// ---- POUs/METS/Common LIB/02_OUTER LIB/Outer FBs/FB_OUTER_ValidationCameraOut.TcPOU
FUNCTION_BLOCK FB_OUTER_ValidationCameraOut
VAR_INPUT
	bDoubleCameraValidationSystemInUse	: BOOL;
	bNewOuterIsProccesing					: BOOL;
	bValidationTimeout						: BOOL;
	bOuterValidation1CameraDone			: BOOL;
	stOuterValidation1CameraStatus	: ST_SCANNER;
	bOuterValidation2CameraDone			: BOOL;
	stOuterValidation2CameraStatus	: ST_SCANNER;

END_VAR
VAR_OUTPUT
	stOuterValidationCameraStatusOut	: ST_SCANNER;
	bOuterValidationDataReady		: BOOL;

END_VAR
VAR
	fbExecute				: R_TRIG;
	aOuterValidationDataReady		: ARRAY [1..2] OF BOOL;
	aCameraNOKStatistic				: ARRAY[1..4] OF INT;
END_VAR

(* rising edge of bExecute *)
fbExecute(CLK:= bNewOuterIsProccesing);

(* move CaseData *)
IF fbExecute.Q = TRUE THEN

	MEMSET(ADR(stOuterValidationCameraStatusOut), 16#00, SIZEOF(stOuterValidationCameraStatusOut));
	bOuterValidationDataReady	:= FALSE;

	aOuterValidationDataReady[1] := FALSE;
	aOuterValidationDataReady[2] := FALSE;
END_IF

IF bOuterValidation1CameraDone OR NOT bDoubleCameraValidationSystemInUse THEN aOuterValidationDataReady[1] := TRUE;	END_IF
IF bOuterValidation2CameraDone THEN aOuterValidationDataReady[2] := TRUE;	END_IF

IF bValidationTimeout	OR
	(bNewOuterIsProccesing AND	aOuterValidationDataReady[1] AND aOuterValidationDataReady[2]) THEN


	IF stOuterValidation1CameraStatus.sImageData.aCodeData[1].strDataString <> '' AND
			 stOuterValidation2CameraStatus.sImageData.aCodeData[1].strDataString = '' THEN

		stOuterValidationCameraStatusOut := stOuterValidation1CameraStatus;

		aCameraNOKStatistic[1] := aCameraNOKStatistic[1] + 1;

	ELSIF stOuterValidation1CameraStatus.sImageData.aCodeData[1].strDataString = '' AND
			 stOuterValidation2CameraStatus.sImageData.aCodeData[1].strDataString <> '' THEN

		stOuterValidationCameraStatusOut := stOuterValidation2CameraStatus;

		aCameraNOKStatistic[2] := aCameraNOKStatistic[2] + 1;

	ELSIF stOuterValidation1CameraStatus.sImageData.aCodeData[1].strDataString <> '' AND
			 stOuterValidation2CameraStatus.sImageData.aCodeData[1].strDataString <> '' AND
			stOuterValidation1CameraStatus.sImageData.aCodeData[1].strDataString = stOuterValidation2CameraStatus.sImageData.aCodeData[1].strDataString THEN

		stOuterValidationCameraStatusOut := stOuterValidation2CameraStatus;

		aCameraNOKStatistic[3] := aCameraNOKStatistic[3] + 1;

	ELSIF stOuterValidation1CameraStatus.sImageData.aCodeData[1].strDataString <> '' AND
			 stOuterValidation2CameraStatus.sImageData.aCodeData[1].strDataString <> '' AND
			stOuterValidation1CameraStatus.sImageData.aCodeData[1].strDataString <> stOuterValidation2CameraStatus.sImageData.aCodeData[1].strDataString THEN

		stOuterValidationCameraStatusOut := stOuterValidation2CameraStatus;
		stOuterValidationCameraStatusOut.sImageData.aCodeData[1].strDataString	:= cCODE_OVERWIRTTEN;

		aCameraNOKStatistic[4] := aCameraNOKStatistic[4] + 1;

	END_IF

	aOuterValidationDataReady[1] := FALSE;
	aOuterValidationDataReady[2] := FALSE;

	bOuterValidationDataReady := TRUE;
END_IF

END_FUNCTION_BLOCK

// ---- POUs/METS/Common LIB/02_OUTER LIB/Outer FBs/FB_OUTER_WriteErrorTable.TcPOU
(* logs data for failed Outers *)
FUNCTION_BLOCK FB_OUTER_WriteErrorTable
VAR_INPUT
	bExecute									: BOOL;			(* set TRUE to scan arrOuterStatus for invalid Outers *)
	bClearData									: BOOL;			(* set TRUE to clear data for invalid Outers *)
	nOpMode									: INT;
	aConfPackCodeInPosition					: ARRAY[1..2] OF T_PACK_Barcode;
	stOuterPackCodeDataNotFound			: ST_RejectItems;
END_VAR
VAR_IN_OUT
	nErrorIndex			: INT;			(* index of Error Outer to be displayed *)
	aOuterStatus			: ARRAY[1..cMAX_OUTER_STATUS_QUEUE] OF ST_OUTER_Status;	(* Outer status array *)
	aErrorOuters			: ARRAY[1..cMAX_OUTER_STATUS_QUEUE] OF ST_OUTER_Status; (* status for last 50 failed Outers *)
END_VAR
VAR_OUTPUT
	bDone				: BOOL;			(* TRUE = OAC action complete *)
	bBusy				: BOOL;			(* TRUE = OAC action in progress *)
	bError				: BOOL;			(* TRUE = OAC action error *)
	nErrorID				: UDINT;		(* error ID *)
	(*bFileInitOK			: BOOL;*)
	nErrorOuters			: UDINT;		(* Outers added to Error list *)
	stErrorOuter			: ST_OUTER_Status; (* last Outer added to arrErrorOuters *)
END_VAR
VAR
	fbExecute				: R_TRIG;
	fbClearData			: R_TRIG;
	eState				: E_OUTER_State;

	nPackIndex			: T_PositiveINT;
	nOuterIndex			: T_PositiveINT;
	(*nMaxOuterIndex		: INT;*)
	nPackStatusIndex		: T_PositiveINT;

	nDupPackChk			: T_PositiveINT;
	nCheckDoubleFail		: T_PositiveINT;
END_VAR

(* monitor bExecute and bClearData for rising edge *)
fbExecute(CLK := bExecute);
fbClearData(CLK := bClearData);

IF fbClearData.Q = TRUE THEN

	(* clear Outer error data *)
	MEMSET(ADR(aErrorOuters), 16#00, SIZEOF(aErrorOuters));
	(*nErrorIndex := 1;*)
END_IF

CASE eState OF

	(* monitor OAC buffer *)
	E_OUTER_IDLE:

		(* rising edge of bExceute *)
		IF fbExecute.Q = TRUE THEN

			(* update outputs *)
			bDone := FALSE;
			bBusy := TRUE;
			bError := FALSE;
			nErrorID := 0;

			(* clear total and reset flag *)
			nErrorOuters := 0;
			(*nMaxOuterIndex := UDINT_TO_INT(SIZEOF(aOuterStatus) / SIZEOF(aOuterStatus[1]));*)


			eState := E_OUTER_SCAN;

		(* bExecute has been reset *)
		ELSIF bExecute = FALSE THEN

			(* reset outputs *)
			bDone := FALSE;
			bBusy := FALSE;
			bError := FALSE;
			nErrorID := 0;
		END_IF


	(* check for Outers that have failed validation *)
	E_OUTER_SCAN:

		(* scan arrStatusArray *)
		FOR nOuterIndex := 1 TO cMAX_OUTER_STATUS_QUEUE DO

			(* CodingAndTrackingMode  > 0 indicates Outer data present *)
			IF aOuterStatus[nOuterIndex].stOACData.CodingAndTrackingMode > 0  AND nOpMode >= 7 THEN

				(* OAC file write error OR validation failed AND data has not been written to ErrorOAC file *)

				(*IF (aOuterStatus[nOuterIndex].nStatus.11  OR aOuterStatus[nOuterIndex].nStatus.13 ) AND NOT aOuterStatus[nOuterIndex].nStatus.14  THEN*)
				IF aOuterStatus[nOuterIndex].nStatus.11 AND NOT aOuterStatus[nOuterIndex].nStatus.14  THEN

					(* update status and log ID for last Outer added *)
					aOuterStatus[nOuterIndex].nStatus.14 := TRUE;

					(* shift arrOACData from [1..49] to [2..50] and move stOACData to arrOACData [1] *)
					MEMMOVE(ADR(aErrorOuters[2]), ADR(aErrorOuters[1]), SIZEOF(aErrorOuters) - SIZEOF(aErrorOuters[1]));
					MEMMOVE(ADR(aErrorOuters[1]), ADR(aOuterStatus[nOuterIndex]), SIZEOF(aErrorOuters[1]));

					IF	aErrorOuters[1].stOACData.OuterRejectID = stOuterPackCodeDataNotFound.nRejectID THEN

						aErrorOuters[1].stOACData.AggregationCodes[1] := aConfPackCodeInPosition[1];
						aErrorOuters[1].stOACData.AggregationCodes[2] := aConfPackCodeInPosition[2];
					END_IF

					(*IF aErrorOuters[1].nStatus.10 AND aErrorOuters[1].nStatus.13 THEN
						aErrorOuters[1].stOACData.OuterRejectCode	:= CONCAT(aErrorOuters[1].stOACData.OuterRejectCode, ' - OAC File Write Error');
					END_IF*)

					(* update counter and set flag to update error file *)
					stErrorOuter := aErrorOuters[1];
					nErrorOuters := nErrorOuters + 1;

					(*AS mod test for previous existence of the failed outer with the same code(s) failed*)
					(*only check if a pack code is missing!*)
					nCheckDoubleFail := 0;
					FOR nPackIndex := 1 TO cMAX_PACKS_PER_OUTER DO
						IF aErrorOuters[1].stOACData.PackCode[nPackIndex] = '' THEN
							nCheckDoubleFail := nCheckDoubleFail+1;
						END_IF
					END_FOR
					IF (nCheckDoubleFail > 0) AND (nCheckDoubleFail < aErrorOuters[1].stOACData.NumberOfPacks) AND nOpMode = 11 AND NOT(aErrorOuters[1].nStatus.15) THEN
						FOR nDupPackChk := 2 TO cMAX_OUTER_STATUS_QUEUE DO
							FOR nPackStatusIndex :=1 TO cMAX_PACKS_PER_OUTER DO
								IF aErrorOuters[1].stOACData.PackCode[nPackStatusIndex] = aErrorOuters[nDupPackChk].stOACData.PackCode[nPackStatusIndex] THEN
										(*Using status 15 for signifying that an outer has failed more than once for the same reason*)
										aErrorOuters[1].nStatus.15 := TRUE;
										aErrorOuters[nDupPackChk].nStatus.15 := TRUE;
									EXIT;
								END_IF
							END_FOR
						END_FOR
					END_IF

					(* update nErrorIndex so that it moves with Outer if new data is added to arrErrorOuter *)
					nErrorIndex := nErrorIndex + 1;
					EXIT;
				END_IF
			END_IF
		END_FOR

		(* end of arrOuterStatus reached *)
		IF nOuterIndex > cMAX_OUTER_STATUS_QUEUE THEN

			eState := E_OUTER_DONE;

		ELSE

			eState := E_OUTER_SCAN;

		END_IF

	(* OAC file complete *)
	E_OUTER_DONE:

		(* update outputs *)
		bDone := TRUE;
		bBusy := FALSE;

		eState := E_OUTER_IDLE;


(* unknown state *)
ELSE

	eState := E_OUTER_IDLE;

	(* reset outputs *)
	bDone := TRUE;
	bBusy := FALSE;
	bError := TRUE;
	nErrorID := 16#FFFFFFFF;

END_CASE

END_FUNCTION_BLOCK

// ---- POUs/METS/Common LIB/02_OUTER LIB/Outer FBs/FB_OUTER_WriteOACLoopDB.TcPOU
(* scan and validate Outers, generate OAC file for new valid Outers *)
FUNCTION_BLOCK FB_OUTER_WriteOACLoopDB
VAR_INPUT
	bExecute					: BOOL;			(* scan for completed Outer *)
	nPacksPerOuter			: INT;
	bExtendedDupCheck		: BOOL;
	nCodingAndTrackingMode	: INT;
	stCTDateTime				: ST_SYSTEM_DateTime;
END_VAR
VAR_IN_OUT
	stOACDataDB					: ST_DB_OACDataCtrl;
	stLastOACDataDB				: ST_DB_OACDataCtrl;
	stCodeInfo_Pack				: ST_CodeInfo;
	stCodeInfo_Outer			: ST_CodeInfo;
	aOuterStatus				: ARRAY[1..cMAX_OUTER_STATUS_QUEUE] OF ST_OUTER_Status;	(* Outer status array *)
	stLastOuterStatus			: ST_OUTER_Status;
	stOuterDataNotFound			: ST_RejectItems;
	stInfeedQueue				: ST_CASE_InfeedQueue;	(* Infeed Conveyor queue *)
END_VAR
VAR_OUTPUT
	bDone				: BOOL;			(* TRUE = validation complete *)
	bBusy				: BOOL;			(* TRUE = validation in progress *)
	bError				: BOOL;			(* TRUE = validation error *)
	nErrorID				: UDINT;		(* error ID *)
	sOACRecordDBName			: T_MaxString;
	stOuterStatus			: ST_OUTER_Status;	(* Outer status *)
	bOACUpdated			: BOOL;
	sCodesAggregatedToOAC	: T_LongSTRING;
END_VAR
VAR
	fbExecute				: R_TRIG;
	tonTimeOut				: TON;
	rtTimeOutExec				: R_TRIG;

	eState					: E_OUTER_State;
	eErrorState					: E_OUTER_State;
	//nMaxOuterIndex		: INT;
	nOuterIndex			: INT;
	nSourceIndex			: INT;
	nInfeedIndex			: INT;

	nCheckIndex : T_PositiveINT;
	nPackIndex : T_PositiveINT;

	eCodeAIType			: E_CodeAIType;

	sBarcode				: T_OUTER_Barcode;

	nOACDataCreated 			: UDINT;
	nOACStoredInDB 			: UDINT;
	nOACFaildInDB				: UDINT;
	nOACUpdatedInDB			: UDINT;

	aDiagOACDataDB				: ARRAY[0..1] OF ST_DB_OACDataCtrl;

	aLocalOuterStatus			: ARRAY[1..10] OF  ST_OUTER_Status;
	nCounter :UDINT;

	nOACLogIndex			: T_PositiveINT;
	sAppendedString				: STRING;
END_VAR

(***************************************TimeOut *******************************************)
(* monitor Busy timeout *)
tonTimeOut( IN:=nSourceIndex <> 0, PT:=cONE_SECOND, Q=>);

rtTimeOutExec(CLK:= tonTimeOut.Q);

IF rtTimeOutExec.Q THEN

	bError := TRUE;
	nErrorID := 100;
	IF nSourceIndex > 0 THEN

		aOuterStatus[nSourceIndex].sDataSourceTracker 	:= 	'TIMEOUT';
		aOuterStatus[nSourceIndex].nStatus.13 := TRUE;

		stLastOuterStatus := aOuterStatus[nSourceIndex];

		sCodesAggregatedToOAC	:= 'TIMEOUT_OUT';
		bOACUpdated	:= TRUE;

	END_IF

	MEMSET(ADR(stOACDataDB), 16#00, SIZEOF(stOACDataDB));
	MEMSET(ADR(stLastOACDataDB), 16#00, SIZEOF(stLastOACDataDB));


	eState := E_OUTER_DONE;
END_IF

(***************************************Execution*******************************************)

(* monitor rising edge of bExecute *)
fbExecute(CLK := bExecute);

(* rising edge of bExecute *)
CASE eState OF

	(* idle *)
	E_OUTER_IDLE:

		(* scan for completed Outer when OAC files are required *)
		IF fbExecute.Q = TRUE THEN

			(* update outputs *)
			bDone := FALSE;
			bBusy := TRUE;
			bError := FALSE;
			nErrorID := 0;

			(* clear outputs *)
			nOACDataCreated 		:= 0;
			nOACStoredInDB 		:= 0;
			nOACFaildInDB			:= 0;

			(* max Outer index *)
			//nMaxOuterIndex := UDINT_TO_INT(SIZEOF(aOuterStatus) / SIZEOF(aOuterStatus[1]));

			eState := E_OUTER_SCAN;

		(* no action required *)
		ELSIF bExecute = FALSE THEN

			(* reset outputs *)
			bDone := FALSE;
			bBusy := FALSE;
			bError := FALSE;
			nErrorID := 0;
		END_IF


	(* scan for completed Outer *)
	E_OUTER_SCAN:

		(* reset index of Outer to be written to OAC file *)
		nSourceIndex 			:= 0;

		sBarcode					:= '';
		bOACUpdated				:= FALSE;

		(* scan aOuterStatus  backward - ensures that oldest Outer will be written first *)
		FOR nOuterIndex := cMAX_OUTER_STATUS_QUEUE TO 1 BY -1 DO

			(* TriggerID > 0 indicates Outer data present -  *)
			IF aOuterStatus[nOuterIndex].nTriggerID > 0 AND
				aOuterStatus[nOuterIndex].stOACData.CodingAndTrackingMode >= 7 AND
				(aOuterStatus[nOuterIndex].nStatus.10  OR
					(aOuterStatus[nOuterIndex].nStatus.11 AND aOuterStatus[nOuterIndex].nStatus.14)) AND
				NOT aOuterStatus[nOuterIndex].nStatus.12 AND
				NOT aOuterStatus[nOuterIndex].nStatus.13 THEN

				(* log index of Outer requiring OAC file *)
				nSourceIndex := nOuterIndex;
				EXIT;
			END_IF
		END_FOR

		(* Outer found requiring OAC file to be written *)
		IF nSourceIndex > 0 THEN

			(* copy Outer data from aOuterStatus *)
			stOuterStatus := aOuterStatus[nSourceIndex];

			nOACDataCreated := nOACDataCreated +1;

			IF	bExtendedDupCheck AND aOuterStatus[nSourceIndex+1].nStatus.12 AND nSourceIndex <  cMAX_OUTER_STATUS_QUEUE  THEN
				(* for all other Packs in Outer *)
				FOR  nPackIndex :=1 TO cMAX_PACKS_PER_OUTER DO
	
					IF stOuterStatus.stOACData.PackCodeStatus[nPackIndex].5 OR stOuterStatus.stOACData.PackCodeStatus[nPackIndex].6 THEN

						FOR nCheckIndex :=1 TO cMAX_PACKS_PER_OUTER DO

							IF stOuterStatus.stOACData.PackCode[nPackIndex] = aOuterStatus[nSourceIndex+1].stOACData.PackCode[nCheckIndex] THEN

								stOuterStatus.nStatus.22 := TRUE;
								stOuterStatus.sDataSourceTracker  := 'OUT_DUPLIC';

								aOuterStatus[nSourceIndex+1].nStatus.22 := TRUE;
								aOuterStatus[nSourceIndex+1].sDataSourceTracker  := 'OUT_DUPLIC';

								EXIT;
							END_IF
						END_FOR
						EXIT;
					END_IF
				END_FOR
			END_IF

			IF aOuterStatus[nSourceIndex+1].nStatus.22 AND stOuterStatus.nStatus.22  AND nSourceIndex <  cMAX_OUTER_STATUS_QUEUE  THEN

				FOR nInfeedIndex:=1 TO stInfeedQueue.nIndex DO 
					IF stInfeedQueue.aOuter[nInfeedIndex].Barcode = aOuterStatus[nSourceIndex+1].stOACData.Barcode 	AND 
						aOuterStatus[nSourceIndex+1].stOACData.Barcode <> ''				 						THEN
						
						stInfeedQueue.aOuter[nInfeedIndex].DataSource 		:= 'B_22';
						stInfeedQueue.aOuter[nInfeedIndex].OuterRejectCode 	:= stOuterDataNotFound.sMetsDisplayCode;
						stInfeedQueue.aOuter[nInfeedIndex].OuterRejectID	:= stOuterDataNotFound.nRejectID;
					END_IF
				END_FOR
				
				stLastOACDataDB.stOACStatusDB	:= aOuterStatus[nSourceIndex+1];
				stLastOACDataDB.bBlockRecord	:= TRUE;
				stLastOACDataDB.bUpdateDataReq 	:= TRUE;

				eState := E_OUTER_UPDATEDATA;
			ELSE
				eState := E_OUTER_WRITEDATA;
			END_IF
		ELSE
			eState := E_OUTER_DONE;
		END_IF

	E_OUTER_UPDATEDATA:

		IF	stLastOACDataDB.bDone	THEN

			IF NOT  stLastOACDataDB.bError THEN

				nOACUpdatedInDB := nOACUpdatedInDB +1;
			ELSE
				bError := TRUE;
				nErrorID := stLastOACDataDB.nErrorID;
				eErrorState := eState;
			END_IF

			aDiagOACDataDB[1]	:= stLastOACDataDB;

			eState := E_OUTER_WRITEDATA;
		END_IF


	E_OUTER_WRITEDATA:

		IF F_InvalidateASCIIChar(F_CODE_GetItem(stOuterStatus.stOACData.Barcode, eCodeAIType.SerialCode, stCodeInfo_Outer)) >	0 	THEN

			stOuterStatus.sDataSourceTracker  := 'BRCD_INVAL';
			stOuterStatus.nStatus.22 := TRUE;
		ELSE
			stOACDataDB.sFileCodeName	:= F_CodeToHex(F_CODE_GetItem(stOuterStatus.stOACData.Barcode , eCodeAIType.SerialCode, stCodeInfo_Outer));
		END_IF

		IF stOuterStatus.nStatus.22 THEN
			stOACDataDB.bBlockRecord		:= TRUE;
		END_IF
		stOACDataDB.stOACStatusDB			:= stOuterStatus;
		stOACDataDB.bCreateDataReq			:= TRUE;

(*place for HectorDB block*)

		IF	stOACDataDB.bDone	THEN

			sOACRecordDBName	:= stOACDataDB.sFileCodeName;

			IF NOT  stOACDataDB.bError THEN

				(* count OAC records stored *)
				nOACStoredInDB := nOACStoredInDB + 1;
				(* update sOuterStatus - OAC record written OK *)
				stOuterStatus.nStatus.12 := TRUE;

			ELSE
				bError := TRUE;
				nErrorID := stOACDataDB.nErrorID;
				nOACFaildInDB := nOACFaildInDB + 1;
				(* update sOuterStatus - OAC file write error *)
				stOuterStatus.stOACData.OuterCodeStatus.6 := TRUE;
				stOuterStatus.nStatus.13 := TRUE;
				eErrorState := eState;
			END_IF

			aDiagOACDataDB[0]	:= stOACDataDB;

			eState := E_OUTER_UPDATESTATUS;

		END_IF

	(* update Outer status *)
	E_OUTER_UPDATESTATUS:

		MEMSET(ADR(stOACDataDB), 16#00, SIZEOF(stOACDataDB));		(*or moved to te execution part at the begining*)
		MEMSET(ADR(stLastOACDataDB), 16#00, SIZEOF(stLastOACDataDB));		(*or moved to te execution part at the begining*)

		(* move stOuterStatus data back to shift reg *)
		FOR nOuterIndex := cMAX_OUTER_STATUS_QUEUE TO 1 BY -1 DO

			(* matching nTriggerID found *)
			IF aOuterStatus[nOuterIndex].nTriggerID = stOuterStatus.nTriggerID AND
				NOT aOuterStatus[nOuterIndex].nStatus.12 AND NOT aOuterStatus[nOuterIndex].nStatus.13 THEN


				nCounter := nCounter +1;
		(*!*)	stLastOuterStatus :=stOuterStatus;
				MEMMOVE(ADR(aLocalOuterStatus[2]), ADR(aLocalOuterStatus[1]), SIZEOF(aLocalOuterStatus)-SIZEOF(aLocalOuterStatus[1]));
				aLocalOuterStatus[1] :=stLastOuterStatus;

				(* move updated Outer data to shift reg *)
				aOuterStatus[nOuterIndex] := stOuterStatus;

				sAppendedString			:= '';
				sCodesAggregatedToOAC	:= '';
				
				sCodesAggregatedToOAC := F_CONCAT3(aOuterStatus[nOuterIndex].stOACData.OuterRejectCode,' - ',  F_CODE_GetItem(aOuterStatus[nOuterIndex].stOACData.Barcode, eCodeAIType.SerialCode, stCodeInfo_Outer));
				sCodesAggregatedToOAC := F_CONCAT6(sCodesAggregatedToOAC,'	[', RIGHT(aOuterStatus[nOuterIndex].stOACData.AggregationCodes[1],7),']:[',RIGHT(aOuterStatus[nOuterIndex] .stOACData.AggregationCodes[2],7),']');

				FOR nOACLogIndex := 1 TO MIN(nPacksPerOuter ,cMAX_PACKS_PER_OUTER) BY 1 DO
					//sCodesAggregatedToOAC :=F_LongCONCAT(sCodesAggregatedToOAC, '     ');
					//sCodesAggregatedToOAC := F_LongCONCAT(sCodesAggregatedToOAC, RIGHT(F_CODE_GetItem(aOuterStatus[nOuterIndex] .stOACData.PackCode[nOACLogIndex], eCodeAIType.SerialCode, stCodeInfo_Pack),7));
				
					CONCAT2(ADR(sCodesAggregatedToOAC), ADR('   '), ADR(sCodesAggregatedToOAC), SIZEOF(sCodesAggregatedToOAC));
		
					sAppendedString := RIGHT(F_CODE_GetItem(aOuterStatus[nOuterIndex].stOACData.PackCode[nOACLogIndex], eCodeAIType.SerialCode, stCodeInfo_Pack),7);
					CONCAT2(ADR(sCodesAggregatedToOAC), ADR(sAppendedString), ADR(sCodesAggregatedToOAC), SIZEOF(sCodesAggregatedToOAC));

				END_FOR

				bOACUpdated := TRUE;
				EXIT;
			END_IF
		END_FOR

		eState := E_OUTER_SCAN;

	(* OAC file complete *)
	E_OUTER_DONE:

		(* update outputs *)
		bDone := TRUE;
		bBusy := FALSE;

		eState := E_OUTER_IDLE;


(* unknown state *)
ELSE

	eState := E_OUTER_IDLE;
END_CASE

END_FUNCTION_BLOCK

// ---- POUs/METS/Common LIB/02_OUTER LIB/Outer Functions/F_OUTER_GetRejectReasonFSS.TcPOU
FUNCTION F_OUTER_GetRejectReasonFSS : T_FSS_RejecCode
VAR_INPUT
	sRejectReasonME			:	STRING(255);
	stOuterRejectReasons	: ST_RejectReasonsForOuter;
END_VAR
VAR
	sRejectReasonFSS:	T_FSS_RejecCode;
END_VAR

IF sRejectReasonME = 'OK' THEN
	sRejectReasonFSS := '';

ELSIF sRejectReasonME = '' THEN
	sRejectReasonFSS := stOuterRejectReasons.stUnknownOuterReject.sFssSendCode;

ELSIF FIND(sRejectReasonME, stOuterRejectReasons.stOuterBarcodeGtinError.sMetsSearchCode) > 0 THEN
	sRejectReasonFSS := stOuterRejectReasons.stOuterBarcodeGtinError.sFssSendCode;

ELSIF FIND(sRejectReasonME, stOuterRejectReasons.stOuterBarcodeRskuError.sMetsSearchCode) > 0 THEN
	sRejectReasonFSS := stOuterRejectReasons.stOuterBarcodeRskuError.sFssSendCode;

ELSIF FIND(sRejectReasonME, stOuterRejectReasons.stOuterCodeSerialError.sMetsSearchCode) > 0 THEN
	sRejectReasonFSS := stOuterRejectReasons.stOuterCodeSerialError.sFssSendCode;

ELSIF FIND(sRejectReasonME, stOuterRejectReasons.stOuterBarcodeInvalidLength.sMetsSearchCode) > 0 THEN
	sRejectReasonFSS := stOuterRejectReasons.stOuterBarcodeInvalidLength.sFssSendCode;

ELSIF FIND(sRejectReasonME, stOuterRejectReasons.stOuterBarcodeNotRead.sMetsSearchCode) > 0 THEN
	sRejectReasonFSS := stOuterRejectReasons.stOuterBarcodeNotRead.sFssSendCode;

ELSIF FIND(sRejectReasonME, stOuterRejectReasons.stOuterBarcodeDuplicate.sMetsSearchCode) > 0 THEN
	sRejectReasonFSS := stOuterRejectReasons.stOuterBarcodeDuplicate.sFssSendCode;

ELSIF FIND(sRejectReasonME,stOuterRejectReasons.stOuterDataNotFound.sMetsSearchCode) > 0 THEN
	sRejectReasonFSS := stOuterRejectReasons.stOuterDataNotFound.sFssSendCode;

ELSIF FIND(sRejectReasonME, stOuterRejectReasons.stOuterGeneralCodeError.sMetsSearchCode) > 0 THEN
	sRejectReasonFSS := stOuterRejectReasons.stOuterGeneralCodeError.sFssSendCode;

ELSIF FIND(sRejectReasonME, stOuterRejectReasons.stOuterTimeOutValidation.sMetsSearchCode) > 0 THEN
	sRejectReasonFSS := stOuterRejectReasons.stOuterTimeOutValidation.sFssSendCode;

ELSIF FIND(sRejectReasonME, stOuterRejectReasons.stOuterDuplicatedPackCodesFound.sMetsSearchCode) > 0 THEN
	sRejectReasonFSS := stOuterRejectReasons.stOuterDuplicatedPackCodesFound.sFssSendCode;

ELSIF FIND(sRejectReasonME, stOuterRejectReasons.stOuterPackCodeDataNotFound.sMetsSearchCode) > 0 THEN
	sRejectReasonFSS := stOuterRejectReasons.stOuterPackCodeDataNotFound.sFssSendCode;

ELSIF FIND(sRejectReasonME, stOuterRejectReasons.stOuterConfirmCodeNotRead.sMetsSearchCode) > 0 THEN
	sRejectReasonFSS := stOuterRejectReasons.stOuterConfirmCodeNotRead.sFssSendCode;

ELSIF FIND(sRejectReasonME, stOuterRejectReasons.stOuterPackCodeInvalid.sMetsSearchCode) > 0 THEN
	sRejectReasonFSS := stOuterRejectReasons.stOuterPackCodeInvalid.sFssSendCode;

ELSIF FIND(sRejectReasonME, stOuterRejectReasons.stOuterPackCodeNotRead.sMetsSearchCode) > 0 THEN
	sRejectReasonFSS := stOuterRejectReasons.stOuterPackCodeNotRead.sFssSendCode;

ELSIF FIND(sRejectReasonME, stOuterRejectReasons.stOuterQAReject.sMetsSearchCode) > 0 THEN
	sRejectReasonFSS := stOuterRejectReasons.stOuterQAReject.sFssSendCode;

ELSIF FIND(sRejectReasonME, stOuterRejectReasons.stOuterPackCodeDBError.sMetsSearchCode) > 0 THEN
	sRejectReasonFSS := stOuterRejectReasons.stOuterPackCodeDBError.sFssSendCode;

ELSIF FIND(sRejectReasonME, stOuterRejectReasons.stOuterBarcodeDBError.sMetsSearchCode) > 0 THEN
	sRejectReasonFSS := stOuterRejectReasons.stOuterBarcodeDBError.sFssSendCode;

ELSIF FIND(sRejectReasonME, stOuterRejectReasons.stOuterCodesBrandSpecError.sMetsSearchCode) > 0 THEN
	sRejectReasonFSS := stOuterRejectReasons.stOuterCodesBrandSpecError.sFssSendCode;

ELSE
	sRejectReasonFSS := stOuterRejectReasons.stUnknownOuterReject.sFssSendCode;
END_IF

F_OUTER_GetRejectReasonFSS := sRejectReasonFSS;

END_FUNCTION

// ---- POUs/METS/Common LIB/02_OUTER LIB/Outer Functions/F_OUTER_HexToBarcode.TcPOU
FUNCTION F_OUTER_HexToBarcode : STRING(255)
VAR_INPUT
	strSerialCodeInHex	: STRING(255);
END_VAR
VAR

	nBarcodeLen		: INT;
	nCharIndex		: INT;
	strCharInHex			: STRING(2);
	nAsciiCode			:BYTE;
	strChar			: STRING(2);
END_VAR

(* reset output *)
F_OUTER_HexToBarcode := '';

(* length of strPackCode *)
nBarcodeLen := LEN(strSerialCodeInHex);

(* strPackCode contains data *)
IF nBarcodeLen > 0 THEN

	(* check each char in the code *)
	FOR nCharIndex := 1 TO nBarcodeLen BY 2 DO

		(* get char from string *)
		strCharInHex := MID(strSerialCodeInHex, 2, nCharIndex);
		HEXSTR_TO_DATA(strCharInHex, ADR(nAsciiCode), SIZEOF(nAsciiCode));
		strChar := F_ToCHR(nAsciiCode);
		F_OUTER_HexToBarcode := CONCAT(F_OUTER_HexToBarcode, strChar);
	END_FOR
END_IF

END_FUNCTION

// ---- POUs/METS/Common LIB/02_OUTER LIB/Outer Functions/F_OUTER_ProgNumberMap.TcPOU
FUNCTION F_OUTER_ProgNumberMap : BOOL

VAR
	nPackIndex			: INT;
END_VAR
(*All VAR_IN_OUT variables have been moved to the end of the declaration due to compatibility reasons*)
VAR_IN_OUT
	stImageData				: ST_SCANNER_ImageData;	(* scanner response data *)
END_VAR

FOR nPackIndex := 1 TO LIMIT(1, stImageData.nCodesRead, cMAX_CAMERA_PROG_NUMBER) DO

	IF stImageData.aCodeData[nPackIndex].nProgramNo = 0 THEN

		(* code is in upper left quadrant of image *)
		IF stImageData.aCodeData[nPackIndex].fXPos >= 0 THEN

			(* get pack position within Outer *)
			stImageData.aCodeData[nPackIndex].nProgramNo := 1;

		(* code is in lower left quadrant of image *)
		ELSIF stImageData.aCodeData[nPackIndex].fXPos < 0 THEN

			(* get pack position within Outer *)
			stImageData.aCodeData[nPackIndex].nProgramNo := 2;
		END_IF
	END_IF
END_FOR

END_FUNCTION

// ---- POUs/METS/Common LIB/04_CASE LIB/Case FBs/FB_CASE_AddOACDataDBLoop.TcPOU
FUNCTION_BLOCK FB_CASE_AddOACDataDBLoop
VAR_INPUT
	bExecute					: BOOL;			(* scan for valid Outer in arrOuterStatus *)
	bStopOnInvalidCode		: BOOL;						(* set TRUE to give alarm if an invalid code is detected *)
	//bFileReadOnly				: BOOL;
	bATTPModeEnable			: BOOL;
	//sLocalOACPath				: T_FolderPath;	(* TEMP folder path *)
	stCTDateTime				: ST_SYSTEM_DateTime;	(* CaseTrace date/time structure *)
	stOuterDataNotFound		: ST_RejectItems;
END_VAR
VAR_IN_OUT
	stOACDataDB					: ST_DB_OACDataCtrl;
	stCodeInfo_Outer			: ST_CodeInfo;
	stProductInstruction			: ST_PCM_Status;
	aOuterStatus				: ARRAY[1..cMAX_OUTER_STATUS_QUEUE] OF ST_OUTER_Status;	(* Outer status array *)
	stInfeedQueue				: ST_CASE_InfeedQueue;	(* Infeed Conveyor queue *)
END_VAR
VAR_OUTPUT
	bDone					: BOOL;			(* TRUE = write OAC file complete *)
	bBusy					: BOOL;			(* TRUE = write OAC file in progress *)
	bError					: BOOL;			(* TRUE = write OAC file error *)
	nErrorID					: UDINT;			(* error ID *)

	nOACFilesRead				: UDINT;
	nReadOACDataFromStructure	: INT;
	nReadOACDataFromFile		: INT;
	nOACFilesFalseRead 		: INT;

	sOACFile					: T_OAC_Filename;
	stOACData				: ST_OAC_Data;
	bScaningActive			: BOOL;
END_VAR
VAR
	fbExecute					: R_TRIG;
	eState					: E_CASE_State;
	eErrorState				: E_CASE_State;
	nOuterIndex				: INT;
	nMaxOuterIndex			: INT;

	sCurrnetInfeedBarcode		: T_MaxString;
	fbReadXMLData			: FB_XmlSrvRead;
	nScanIndex				: INT;

	sOuterTimeStamp				: T_ISO8601Time;
	bOuterMasterListRestored	: BOOL;
	sDataSource				: STRING(4);

	nCounter					: INT;
END_VAR

(* monitor bExecute for rising edge *)
fbExecute(CLK := bExecute);

CASE eState OF

	(* idle state *)
	E_CASE_IDLE:

		(* rising edge of bExecute *)
		IF fbExecute.Q = TRUE THEN

			(* update outputs *)
			bDone := FALSE;
			bBusy := TRUE;
			bError := FALSE;
			nErrorID := 0;

			(* clear outputs *)
			nOACFilesRead := 0;
			sOACFile := '';
			(*MEMSET(ADR(stOACData), 16#00, SIZEOF(stOACData));*)
			sDataSource :='';
			nMaxOuterIndex := UDINT_TO_INT(SIZEOF(aOuterStatus) / SIZEOF(aOuterStatus[1]));

			(*nOuterIndex := 1;*)

			eState := E_CASE_SCANINFEEDQUEUE;

		(* OAC data disabled *)
		ELSIF bExecute = FALSE THEN

			(* reset outputs *)
			bDone := FALSE;
			bBusy := FALSE;
			bError := FALSE;
			nErrorID := 0;

			bScaningActive := FALSE;

		END_IF


	(* scan for missing OAC data *)
	E_CASE_SCANINFEEDQUEUE:

		(* preset next state, will be udpated if an Outer without OAC data is found in Infeed Queue *)
		MEMSET(ADR(stOACData), 16#00, SIZEOF(stOACData));
		eState := E_CASE_DONE;

		(* scan remainder of Infeed Queue *)
		FOR nScanIndex := 1 TO  MIN(stInfeedQueue.nIndex, cMAX_INFEED_QUEUE) DO

			(* OAC data has not been read *)
			IF stInfeedQueue.aOuter[nScanIndex].CodingAndTrackingMode = 0 AND  stInfeedQueue.aOuter[nScanIndex].DataSource = '' THEN

				IF (*stProductInstruction.nOpMode = 7 AND*) NOT stProductInstruction.bEnablePacks (*AND bStopOnInvalidCode*) THEN
					stInfeedQueue.aOuter[nScanIndex].ProductionDate := F_StringWildcard('#YYYYMMDD#', stCTDateTime.sSystemTime);
					stInfeedQueue.aOuter[nScanIndex].ProductionTime := F_StringWildcard('#hhmmss#', stCTDateTime.sSystemTime);
					stInfeedQueue.aOuter[nScanIndex].ProductionTimeOffset := F_SYSTEM_SystemTimeOffsetToHHMM(stCTDateTime.nSystemTimeOffset);

					stInfeedQueue.aOuter[nScanIndex].OuterTimeStamp :=F_SYSTEM_SystemTimeAsISO8601(stCTDateTime.sSystemTime, stCTDateTime.sUTCTimeZoneOffset );
					stInfeedQueue.aOuter[nScanIndex].RetailSKU := stProductInstruction.sRetailSKU;
					stInfeedQueue.aOuter[nScanIndex].OuterMachine.ProductionSite :=  stProductInstruction.sProductionSite;
					stInfeedQueue.aOuter[nScanIndex].OuterMachine.ProductionLine := stProductInstruction.sProductionLine;
					stInfeedQueue.aOuter[nScanIndex].BatchNumber := stProductInstruction.sBatchNumber;
					stInfeedQueue.aOuter[nScanIndex].CodingAndTrackingMode := stProductInstruction.nOpMode;

					stInfeedQueue.aOuter[nScanIndex].DataSource := 'REST';
					stInfeedQueue.aOuter[nScanIndex].OuterRejectCode := 'OK';
					stInfeedQueue.aOuter[nScanIndex].OuterRejectID := 0;

					eState := E_CASE_SCANINFEEDQUEUE;

				ELSE
					sCurrnetInfeedBarcode 	:=	 stInfeedQueue.aOuter[nScanIndex].Barcode ;
					bOuterMasterListRestored 	:= stInfeedQueue.aOuter[nScanIndex].OuterMasterListRestored;
					(*sOuterTimeStamp			:= stInfeedQueue.aOuter[nScanIndex].OuterTimeStamp;*)
					sDataSource :='';
					(* generate OAC file name and clear data for last OAC file *)

					(*sOACFile := F_CONCAT3('OAC_', F_OUTER_BarcodeToHex(sCurrnetInfeedBarcode), '.xml');*)

					IF bTempBlockReadFromStruct THEN
						eState := E_CASE_SCANOUTERS;
					ELSE
						eState := E_CASE_READOACDATA;
					END_IF
				END_IF

				bScaningActive := TRUE;
				EXIT;
			END_IF
		END_FOR

	E_CASE_SCANOUTERS:


		FOR nOuterIndex := 1 TO nMaxOuterIndex DO

			(* TriggerID > 0 indicates Outer data present *)
			IF	 aOuterStatus[nOuterIndex].bLabelApplied 
				AND NOT aOuterStatus[nOuterIndex].nStatus.19 
				AND NOT aOuterStatus[nOuterIndex].nStatus.22 THEN

				IF  aOuterStatus[nOuterIndex].stOACData.Barcode = sCurrnetInfeedBarcode  THEN

					stOACData	 := aOuterStatus[nOuterIndex].stOACData;
					EXIT;
				END_IF
			END_IF
		END_FOR

		IF stOACData.CodingAndTrackingMode > 0 OR stOACData.OuterRejectCode <> '' THEN

			nOACFilesRead := nOACFilesRead + 1;
			sDataSource := 'ST';
			nReadOACDataFromStructure:= nReadOACDataFromStructure + 1;

			eState := E_CASE_UPDATEINFEEDQUEUE;
		ELSE
			eState := E_CASE_READOACDATA;
		END_IF

	(* read data from OAC *)
	E_CASE_READOACDATA:

				stOACDataDB.bReadDataReq		:=TRUE;

				(*stOACDataDB.sFileCodeName		 := F_OUTER_BarcodeToHex(sCurrnetInfeedBarcode);*)

				IF F_InvalidateASCIIChar(F_CODE_GetItem(sCurrnetInfeedBarcode, eCodeAIType.SerialCode, stCodeInfo_Outer)) >	0 	THEN
		
					stOACDataDB.sFileCodeName := '';
				ELSE
					stOACDataDB.sFileCodeName	:= F_CodeToHex(F_CODE_GetItem(sCurrnetInfeedBarcode , eCodeAIType.SerialCode, stCodeInfo_Outer));
				END_IF

				IF stOACDataDB.bDone THEN
					IF NOT stOACDataDB.bError THEN		(* f.ex not found, or DB transaction faild??*)

						IF NOT  stOACDataDB.stOACStatusDB.nStatus.22 THEN

							stOACData := stOACDataDB.stOACStatusDB.stOACData;
							sDataSource := 'DB';
						ELSE
							sDataSource := 'B_22';
						END_IF

						nOACFilesRead := nOACFilesRead + 1;

					ELSE
						bError := TRUE;
						nErrorID := stOACDataDB.nErrorID;
						sDataSource := 'NO_R';

						eErrorState := eState;
					END_IF

					eState := E_CASE_UPDATEINFEEDQUEUE;

				END_IF

	(* update OAC data to Infeed Queue *)
	E_CASE_UPDATEINFEEDQUEUE:

		MEMSET(ADR(stOACDataDB), 16#00, SIZEOF(stOACDataDB));		(*or moved to te execution part at the begining*)

		(* scan Infeed Queue *)
		FOR nScanIndex := 1 TO  MIN(stInfeedQueue.nIndex, cMAX_INFEED_QUEUE) DO

			(* generate OAC file name AND clear data FOR last OAC file *)
				(* Outer is still in same position in Infeed Queue *)
			IF stInfeedQueue.aOuter[nScanIndex].Barcode = sCurrnetInfeedBarcode THEN

				(* copy OAC data into Infeed Queue *)
				IF stOACData.Barcode = sCurrnetInfeedBarcode AND  stOACData.Barcode <> '' THEN
					stInfeedQueue.aOuter[nScanIndex] := stOACData;
				(*In case File read return error and erase stOACData*)
				ELSIF stOACData.Barcode ='' THEN
					stInfeedQueue.aOuter[nScanIndex].Barcode := sCurrnetInfeedBarcode;
					
					IF sDataSource = 'DB' AND sDataSource <> 'B_22' THEN	sDataSource := 'DB_R';	END_IF
				ELSE
					stInfeedQueue.aOuter[nScanIndex].Barcode := sCurrnetInfeedBarcode;
					stInfeedQueue.aOuter[nScanIndex].DataSource := 'MISS';
				END_IF
				(*stInfeedQueue.aOuter[nScanIndex].OuterTimeStamp			:= sOuterTimeStamp;*)
				stInfeedQueue.aOuter[nScanIndex].DataSource 				:= sDataSource;
				stInfeedQueue.aOuter[nScanIndex].OuterMasterListRestored 	:= bOuterMasterListRestored;
				stInfeedQueue.aOuter[nScanIndex].OuterCodeStatus.4 			:= bOuterMasterListRestored;
				
				IF stInfeedQueue.aOuter[nScanIndex].OuterRejectCode = '' THEN
					stInfeedQueue.aOuter[nScanIndex].OuterRejectCode 	:= stOuterDataNotFound.sMetsDisplayCode;
					stInfeedQueue.aOuter[nScanIndex].OuterRejectID		:= stOuterDataNotFound.nRejectID;
				END_IF

				(*Modif outer time stamp to represent moment of adding OCA data in casepacker*)
				IF bATTPModeEnable THEN
					stInfeedQueue.aOuter[nScanIndex].OuterTimeStamp :=F_SYSTEM_SystemTimeAsISO8601(stCTDateTime.sSystemTime, stCTDateTime.sUTCTimeZoneOffset );
				END_IF

				EXIT;
			END_IF
		END_FOR

		eState := E_CASE_SCANINFEEDQUEUE;

	(* done *)
	E_CASE_DONE:

		bScaningActive := FALSE;

		(* update outputs *)
		bBusy := FALSE;
		bDone := TRUE;

		eState := E_CASE_IDLE;


(* unknown state *)
ELSE

	eState := E_CASE_IDLE;
END_CASE

END_FUNCTION_BLOCK

// ---- POUs/METS/Common LIB/04_CASE LIB/Case FBs/FB_CASE_AddOuterToInfeedQ.TcPOU
(* add strOuterBarcode to sInfeedQueue, will not be added if strOuterBarcode already exists *)
FUNCTION_BLOCK FB_CASE_AddOuterToInfeedQ
VAR_INPUT
	bExecute								: BOOL;		(* set TRUE to add Outer barcode to buffer *)
	sOuterBarcode							: T_OUTER_Barcode;	(* 2D barcode from scanner *)
	bMasterListInUse						: BOOL;
	bUseInterimCodeForLastPosition		: BOOL;
	(*bATTPModeEnable			: BOOL;
	stCTDateTime				: ST_SYSTEM_DateTime;	(* CaseTrace date/time structure *)*)
END_VAR
VAR_IN_OUT
	nRestoreCounter								: UDINT;
	stProductInstruction							: ST_PCM_Status;
	stCodeInfo_Intermediate						: ST_CodeInfo;
	stCodeInfo_Outer								: ST_CodeInfo;
	stInfeedQueue							: ST_CASE_InfeedQueue;	(* Infeed Queue *)
END_VAR
VAR_OUTPUT
	bDone			: BOOL;		(* TRUE = complete *)
	bBarcodeAdded	: BOOL;		(* TRUE = Outer barcode added to queue *)
	bBarcodeValid		: BOOL;		(* TRUE = Outer barcode is valid *)
	bBarcodeExists		: BOOL;		(* TRUE = Outer barcode already present in queue *)
	sLastBarcodeAdded	: T_OUTER_Barcode;	(* last Outer barcode added to sInfeedQueue *)
END_VAR
VAR
	fbExecute			: R_TRIG;
	nOuterIndex		: T_PositiveINT;
	//nMaxOuterIndex	: INT;
	eCodeAIType		: E_CodeAIType;
	fbValidateOuter		: FB_CODE_ValidateExplicitCode;

END_VAR

(* rising edge of bExecute *)
fbExecute(CLK:= bExecute);

(* add Outer to sInfeedQueue *)
IF fbExecute.Q = TRUE THEN

	(* reset outputs *)
	bDone := FALSE;
	bBarcodeAdded := FALSE;
	bBarcodeValid := FALSE;
	bBarcodeExists := FALSE;
	sLastBarcodeAdded	:= '';

	(* sOuterBarcode contains data and is different to last Outer barcode added to queue *)
	IF sOuterBarcode <> '' AND sOuterBarcode <> stInfeedQueue.sLastBarcode THEN

		(* InfeedQueue contains Outers *)
		IF stInfeedQueue.nIndex > 0 THEN

			(* scan all Outers in stInfeedQueue *)
			FOR nOuterIndex := 1 TO  MIN(stInfeedQueue.nIndex, cMAX_INFEED_QUEUE)   DO

				(* sOuterBarcode already exists in stInfeedQueue *)
				(*IF stInfeedQueue.sOuter[nOuterIndex].Barcode = sOuterBarcode  AND stInfeedQueue.sOuter[nOuterIndex].OuterMasterListRestored  AND bMasterListInUse THEN*)

				IF stInfeedQueue.aOuter[nOuterIndex].Barcode = sOuterBarcode  AND stInfeedQueue.aOuter[nOuterIndex].OuterMasterListRestored AND bMasterListInUse THEN

					IF nOuterIndex = cMAX_INFEED_QUEUE THEN
						MEMSET(ADR(stInfeedQueue.aOuter[cMAX_INFEED_QUEUE]), 16#00, SIZEOF(stInfeedQueue.aOuter[1]));
					ELSIF nOuterIndex < cMAX_INFEED_QUEUE THEN
						MEMMOVE(ADR(stInfeedQueue.aOuter[nOuterIndex]), ADR(stInfeedQueue.aOuter[nOuterIndex+1]), SIZEOF(stInfeedQueue.aOuter[1]) * F_SafeTo_UDINT(stInfeedQueue.nIndex - nOuterIndex) );
						MEMSET(ADR(stInfeedQueue.aOuter[stInfeedQueue.nIndex]), 0, SIZEOF(stInfeedQueue.aOuter[1]));
					END_IF
					
					stInfeedQueue.nIndex := stInfeedQueue.nIndex - 1;
					nRestoreCounter	:= MAX(0, nRestoreCounter - 1);

				ELSIF  stInfeedQueue.aOuter[nOuterIndex].Barcode = sOuterBarcode THEN

					bBarcodeExists := TRUE;

					EXIT;
				END_IF
			END_FOR
		END_IF

		(* FOR loop completed, no duplicate code found *)
		IF bBarcodeExists = FALSE THEN

			(* max number of Outers in stInfeedQueue *)
			//nMaxOuterIndex := UDINT_TO_INT(SIZEOF(stInfeedQueue.aOuter) / SIZEOF(stInfeedQueue.aOuter[1]));

			(* list of Outers in stInfeedQueue is full *)
			IF stInfeedQueue.nIndex >= cMAX_INFEED_QUEUE THEN

				(* remove 1st Outer from sInfeedQueue and clear data for last Outer *)
				MEMMOVE(ADR(stInfeedQueue.aOuter[1]), ADR(stInfeedQueue.aOuter[2]), SIZEOF(stInfeedQueue.aOuter) - SIZEOF(stInfeedQueue.aOuter[1]));
				MEMSET(ADR(stInfeedQueue.aOuter[cMAX_INFEED_QUEUE]), 16#00, SIZEOF(stInfeedQueue.aOuter[1]));

				(* update stInfeedQueue pointer *)
				stInfeedQueue.nIndex := cMAX_INFEED_QUEUE - 1;
			END_IF

			(* increment stInfeedQueue pointer and add sOuterBarcode *)

			stInfeedQueue.nIndex := LIMIT(0,stInfeedQueue.nIndex + 1,cMAX_INFEED_QUEUE);
			stInfeedQueue.aOuter[stInfeedQueue.nIndex].Barcode := sOuterBarcode;
			stInfeedQueue.aOuter[stInfeedQueue.nIndex].DataSource :='';

			(*Modif outer time stamp to represent moment of adding OCA data in casepacker*)
			(*IF bATTPModeEnable THEN
				stInfeedQueue.aOuter[stInfeedQueue.nIndex].OuterTimeStamp :=F_SYSTEM_SystemTimeAsISO8601(stCTDateTime.sSystemTime, stCTDateTime.sUTCTimeZoneOffset );
			END_IF*)

			(* update outputs *)
			bBarcodeAdded := TRUE;
			stInfeedQueue.sLastBarcode := sOuterBarcode;
			sLastBarcodeAdded := sOuterBarcode;

			fbValidateOuter(	sFullCode := sOuterBarcode,
							stCodeInfo := SEL(bUseInterimCodeForLastPosition, stCodeInfo_Outer, stCodeInfo_Intermediate),
							stProductInstruction := stProductInstruction);

			IF stProductInstruction.nOpMode >= 7 AND fbValidateOuter.bValidationOK THEN

				(* barcode is valid *)
				bBarcodeValid := TRUE;
			END_IF
		END_IF
	END_IF

	bDone := TRUE;

(* bExecute has been reset *)
ELSIF bExecute = FALSE THEN

	(* reset outputs *)
	bDone := FALSE;
	bBarcodeAdded := FALSE;
	(*bBarcodeValid := FALSE;
	bBarcodeExists := FALSE;*)
END_IF

END_FUNCTION_BLOCK

// ---- POUs/METS/Common LIB/08_SOFTWARE LIB/Memory FBs/F_SafeTo_UDINT.TcPOU
FUNCTION F_SafeTo_UDINT : UDINT
VAR_INPUT
	nCovertVar	: Dint;
END_VAR
VAR
END_VAR

F_SafeTo_UDINT := TO_UDINT(MAX(0,nCovertVar));

END_FUNCTION

// ---- POUs/METS/Common LIB/04_CASE LIB/Case FBs/FB_CASE_AddVerifiedCaseBarcode.TcPOU
FUNCTION_BLOCK FB_CASE_AddVerifiedCaseBarcode
VAR_INPUT
	bExecute									: BOOL;
	bClearVerifiedCaseBarcodesQueue										: BOOL;
	sCaseBarcode									: T_CASE_Barcode;		(* image data structure *)
END_VAR
VAR_IN_OUT
	aLastCaseBarcodes				: ARRAY[1..cMAX_LAST_CASE_BARCODES] OF T_CASE_Barcode;
END_VAR
VAR_OUTPUT
	bDone										: BOOL;
END_VAR
VAR
	rtrigExecute: R_TRIG;
END_VAR

rtrigExecute(CLK := bExecute);

IF bClearVerifiedCaseBarcodesQueue THEN
	MEMSET(ADR(aLastCaseBarcodes), 16#00, SIZEOF(aLastCaseBarcodes));
END_IF

IF rtrigExecute.Q AND NOT bClearVerifiedCaseBarcodesQueue THEN
	bDone := FALSE;

	MEMMOVE(ADR(aLastCaseBarcodes[2]), ADR(aLastCaseBarcodes[1]),  SIZEOF(aLastCaseBarcodes) - SIZEOF(aLastCaseBarcodes[1]));
	MEMSET(ADR(aLastCaseBarcodes[1]), 16#00, SIZEOF(aLastCaseBarcodes[1]));

	aLastCaseBarcodes[1] := sCaseBarcode;

	bDone := TRUE;
ELSE
	bDone := FALSE;
END_IF

END_FUNCTION_BLOCK

// ---- POUs/METS/Common LIB/04_CASE LIB/Case FBs/FB_CASE_FindAndDeleteOuter.TcPOU
FUNCTION_BLOCK FB_CASE_FindAndDeleteOuter
VAR_INPUT
	bExecute						: BOOL;
	strPackBarcode					: T_PACK_Barcode;
	strOuterBarcode				: T_OUTER_Barcode;
	stProductInstruction				: ST_PCM_Status;
END_VAR
VAR_IN_OUT
	stInfeedQueue					: ST_CASE_InfeedQueue;
END_VAR
VAR_OUTPUT
	bDone						: BOOL;			(* TRUE = complete *)
END_VAR
VAR
	fbExecute						: R_TRIG;
	nOuterIndex					: INT;
	nPackIndex					: INT;
	nCodeFoundIndex				: INT;
	bCodeFound					: BOOL;
END_VAR

fbExecute (CLK:= bExecute);

IF fbExecute.Q THEN

	FOR nOuterIndex:=1 TO MIN(stInfeedQueue.nIndex, cMAX_INFEED_QUEUE) DO

		IF strOuterBarcode <> '' THEN

			IF strOuterBarcode =  stInfeedQueue.aOuter[nOuterIndex].Barcode THEN
				nCodeFoundIndex := nOuterIndex;
				bCodeFound := TRUE;
				EXIT;
			END_IF

		ELSIF  strPackBarcode <> '' THEN

			FOR nPackIndex:=1 TO MIN(stProductInstruction.nPacksPerOuter, cMAX_PACKS_PER_OUTER) DO
				IF strPackBarcode = stInfeedQueue.aOuter[nOuterIndex].PackCode[nPackIndex] THEN
					nCodeFoundIndex := nOuterIndex;
					bCodeFound := TRUE;
					EXIT;
				END_IF
			END_FOR

		END_IF

		IF bCodeFound THEN
			EXIT;
		END_IF
	END_FOR

	IF bCodeFound AND nCodeFoundIndex <> 0 THEN
		MEMMOVE(ADR(stInfeedQueue.aOuter[nCodeFoundIndex]), ADR(stInfeedQueue.aOuter[nCodeFoundIndex + 1]), SIZEOF(stInfeedQueue.aOuter[1]) * F_SafeTo_UDINT(cMAX_INFEED_QUEUE - nCodeFoundIndex) );
		MEMSET(ADR(stInfeedQueue.aOuter[cMAX_INFEED_QUEUE]), 16#00, SIZEOF(stInfeedQueue.aOuter[cMAX_INFEED_QUEUE]));
		stInfeedQueue.nIndex :=LIMIT(0, stInfeedQueue.nIndex - 1, cMAX_INFEED_QUEUE);
	END_IF

	bDone := TRUE;
ELSE
	nCodeFoundIndex := 0;
	bCodeFound := FALSE;
	bDone := FALSE;
END_IF

END_FUNCTION_BLOCK

// ---- POUs/METS/Common LIB/04_CASE LIB/Case FBs/FB_CASE_FindCaseInQueue.TcPOU
(* find matching BarcodeMasterCase in Case Queue *)
FUNCTION_BLOCK FB_CASE_FindCaseInQueue
VAR_INPUT
	bExecute			: BOOL;			(* set TRUE to add value to buffer *)
	sCaseData			: ST_CAC_Data;	(* case barcode *)
END_VAR
VAR_IN_OUT
	stCaseQueue			: ST_CASE_CaseQueue;	(* case queue structure *)
END_VAR
VAR_OUTPUT
	bDone				: BOOL;			(* TRUE = complete *)
	bCaseNotFound		: BOOL;			(* TRUE = strCaseBarcode not found *)
	bCaseExists			: BOOL;			(* TRUE = strCaseBarcode found *)
	nCaseIndex			: INT;			(* case location in buffer, 0 = not found *)
END_VAR
VAR
	fbExecute			: R_TRIG;
	//nMaxIndex			: UINT;
	nIndex				: INT;
END_VAR
(*
-------------------------------------------------------------------------------------------------
Date		Version	Author	Comments
-------------------------------------------------------------------------------------------------
24/11/2010	1.07.03	PB		CaseBarcodeDateTimeString checked instead of BarcodeMasterCase when searching for matching Case
02/11/2010	1.07.00	PB		Initial release

-------------------------------------------------------------------------------------------------
*)

(* rising edge of bExecute *)
fbExecute(CLK:= bExecute);

(* search for strBarcode in queue *)
IF fbExecute.Q = TRUE THEN

	(* max index of buffer array *)
	//nMaxIndex := UDINT_TO_UINT(SIZEOF(stCaseQueue.aCACData) / SIZEOF(stCaseQueue.aCACData[1]));

	(* scan all cases in queue *)
	FOR nIndex := 1 TO cMAX_CASE_QUEUE DO

		(* case match found *)
		IF stCaseQueue.aCACData[nIndex].Barcode = sCaseData.Barcode THEN

			bCaseExists := TRUE;
			nCaseIndex := nIndex;
			EXIT;
		END_IF
	END_FOR

	bCaseNotFound := NOT bCaseExists;
	bDone := TRUE;

(* bExecute has been reset *)
ELSIF bExecute = FALSE THEN

	(* reset outputs *)
	bDone := FALSE;
	bCaseNotFound := FALSE;
	bCaseExists := FALSE;
	nCaseIndex := 0;
END_IF

END_FUNCTION_BLOCK

// ---- POUs/METS/Common LIB/04_CASE LIB/Case FBs/FB_CASE_LastRowPoisitionBuffer_v2.TcPOU
(* shift  Image Data from fbScaner  *)
FUNCTION_BLOCK FB_CASE_LastRowPoisitionBuffer_v2
VAR_INPUT
	bExecute					: BOOL;
	bReadError				: BOOL;
	nValideIndex				: INT;
	bResetBuffer				: BOOL;
END_VAR
VAR_IN_OUT
	stNewImageData			: ST_SCANNER_ImageData;
END_VAR
VAR_OUTPUT
	bDone					: BOOL;			(* TRUE = complete *)
	stCurrentImageData			: ST_SCANNER_ImageData;
	sCurrentBarcode			: T_OUTER_Barcode;
	sLastOuterBarcode			: T_OUTER_Barcode;				(* last good received barcode *)
END_VAR
VAR
	fbExecute					: R_TRIG;
	aBufforImageData			: ARRAY[0..4] OF ST_SCANNER_ImageData;		(* image data structure *)
END_VAR

(* rising edge of bExecute *)
fbExecute(CLK:= bExecute);

nValideIndex := LIMIT(0, nValideIndex, 4);

IF bResetBuffer	THEN

(* clear source buffer data *)
	MEMSET(ADR(aBufforImageData), 16#00, SIZEOF(aBufforImageData));
END_IF

IF fbExecute.Q = TRUE THEN

	(* shift Image Data one position  *)
	MEMMOVE(ADR(aBufforImageData[1]), ADR(aBufforImageData[0]), SIZEOF(aBufforImageData)-SIZEOF(aBufforImageData[0]));

	IF bReadError THEN
		MEMSET(ADR(aBufforImageData[0]), 16#00 , SIZEOF(aBufforImageData[0]));
	ELSE
		(* copy Image Data to first position *)
		MEMCPY(ADR(aBufforImageData[0]), ADR(stNewImageData), SIZEOF(aBufforImageData[0]));
	END_IF

	sLastOuterBarcode := sCurrentBarcode;

	(* update output *)
	bDone := TRUE;

(* bExecute has been reset *)
ELSIF bExecute = FALSE THEN

	(* clear output *)
	bDone := FALSE;
END_IF

stCurrentImageData := aBufforImageData[nValideIndex];
sCurrentBarcode :=	aBufforImageData[nValideIndex].aCodeData[1].strDataString;

END_FUNCTION_BLOCK

// ---- POUs/METS/Common LIB/04_CASE LIB/Case FBs/FB_CASE_MasterListControl.TcPOU
FUNCTION_BLOCK FB_CASE_MasterListControl
VAR_INPUT
	bEnableMasterlistFillin			: BOOL;
	bCheckMasterList				: BOOL;
	bMasterListBarcodeAdded		: BOOL;
	sLastBarcodeRead				: T_MaxString;
	aMasterList					: ARRAY[0..cMAX_OUTER_STATUS_QUEUE] OF T_MaxString;
END_VAR
VAR_IN_OUT
	stInfeedQueue					: ST_CASE_InfeedQueue;	(* Infeed Convoyer Queue *)
	nRestoreCounter				: UDINT;
END_VAR
VAR
	rtrigUpdateMasterlist			: R_TRIG;
	rtrigFillInMasterlist				: R_TRIG;
	sLastCode						: STRING := '';
	sCurrentCode					: STRING := '';
	sFillinCode					: STRING := '';
	nIndex						: INT;
	nLastCodePos					: INT;
	nCurrentCodePos				: INT;
	nMaxOuterIndex 				: INT;
	nOuterIndex					: INT;
	bBarcodeExists 				: BOOL;
END_VAR

IF NOT  bEnableMasterlistFillin THEN
	RETURN;
END_IF

rtrigFillInMasterlist(CLK:=bCheckMasterList AND bMasterListBarcodeAdded);

IF rtrigFillInMasterlist.Q THEN
	sCurrentCode := sLastBarcodeRead;
	bBarcodeExists := FALSE;

	IF (sCurrentCode <> '') AND (sLastCode <> '') THEN
		(*findLastCode*)
		nLastCodePos := -1;
		FOR nIndex := 0 TO cMAX_OUTER_STATUS_QUEUE DO
			IF sLastCode = aMasterList[nIndex] THEN
				nLastCodePos := nIndex;
				EXIT;
			END_IF
		END_FOR

		(*findCurrentCode*)
		nCurrentCodePos := -1;
		FOR nIndex := 0 TO cMAX_OUTER_STATUS_QUEUE DO
			IF sCurrentCode = aMasterList[nIndex] THEN
				nCurrentCodePos :=nIndex;
				EXIT;
			END_IF
		END_FOR

		sFillinCode := '';
		IF (nLastCodePos >= 0) AND (nCurrentCodePos >= 0) AND (nLastCodePos - nCurrentCodePos  = 2) THEN
			sFillinCode := aMasterList[nCurrentCodePos+1];


	(* scan all Outers in sInfeedQueue *)
			FOR nOuterIndex := 1 TO  MIN(stInfeedQueue.nIndex, cMAX_INFEED_QUEUE) DO
				(* strOuterBarcode already exists in sInfeedQueue *)
				IF stInfeedQueue.aOuter[nOuterIndex].Barcode = sFillinCode THEN
					bBarcodeExists := TRUE;
					EXIT;
				END_IF
			END_FOR

			IF sFillinCode <> '' AND NOT bBarcodeExists THEN
				(*Create a space in the infeed queue and insert*)
				(* max number of Outers in sInfeedQueue *)
				nMaxOuterIndex := UDINT_TO_INT(SIZEOF(stInfeedQueue.aOuter) / SIZEOF(stInfeedQueue.aOuter[1]));

				(* list of Outers in sInfeedQueue is full so drop one off the end to create space*)
				IF stInfeedQueue.nIndex >= nMaxOuterIndex THEN

					(* remove 1st Outer from sInfeedQueue and clear data for last Outer *)
					MEMMOVE(ADR(stInfeedQueue.aOuter[1]), ADR(stInfeedQueue.aOuter[2]), SIZEOF(stInfeedQueue.aOuter) - SIZEOF(stInfeedQueue.aOuter[1]));
					MEMSET(ADR(stInfeedQueue.aOuter[nMaxOuterIndex]), 16#00, SIZEOF(stInfeedQueue.aOuter[1]));

					(* update sInfeedQueue pointer *)
					stInfeedQueue.nIndex := nMaxOuterIndex - 1;
				END_IF

				(*put in a gap*)
				MEMMOVE(ADR(stInfeedQueue.aOuter[stInfeedQueue.nIndex+1]), ADR(stInfeedQueue.aOuter[stInfeedQueue.nIndex]), SIZEOF(stInfeedQueue.aOuter[1]));
				MEMSET(ADR(stInfeedQueue.aOuter[stInfeedQueue.nIndex]), 16#00, SIZEOF(stInfeedQueue.aOuter[1]));

				(*insert our filled in outer barcode*)

				stInfeedQueue.aOuter[stInfeedQueue.nIndex].Barcode := sFillInCode;

				stInfeedQueue.aOuter[stInfeedQueue.nIndex].OuterMasterListRestored := TRUE;
				stInfeedQueue.aOuter[stInfeedQueue.nIndex].OuterCodeStatus.4 := TRUE;
				nRestoreCounter	:= nRestoreCounter + 1;

				(*increment queue count*)
				stInfeedQueue.nIndex := LIMIT(0,stInfeedQueue.nIndex + 1,cMAX_INFEED_QUEUE);
			END_IF
		END_IF

	END_IF

	sLastCode := sCurrentCode;
END_IF

END_FUNCTION_BLOCK

// ---- POUs/METS/Common LIB/04_CASE LIB/Case FBs/FB_CASE_MoveFailedCAC.TcPOU
(* move failded CaC dato into Failed Cac *)
FUNCTION_BLOCK FB_CASE_MoveFailedCAC
VAR_INPUT
	bExecute 						: BOOL;		(* set TRUE to move Outers *)
	stPrintCACData				: ST_CAC_Data;
	stCTDateTime					: ST_SYSTEM_DateTime;	(* CaseTrace date/time structure *)
	(*stCodeInfo_Case		: ST_CodeInfo;*)
END_VAR
VAR_IN_OUT
	aFailedCACData				: ARRAY[1..cMAX_FAILED_CASE_QUEUE] OF ST_CAC_Data;	(* array of failed CAC data *)
	aFailedCACDataHMI			: ARRAY[1..cMAX_FAILED_CASE_QUEUE] OF ST_HMI_CAC_Data;	(* array of failed CAC data *)
	stQaseQueueDataHMI			: ST_HMI_CAC_Data;
END_VAR
VAR_OUTPUT
	bDone: BOOL;
END_VAR
VAR
	fbExecute						: R_TRIG;
	nIndexOuter					:INT;
	nIndexPack					:INT;
END_VAR

(* rising edge of bExecute *)
fbExecute(CLK:= bExecute);

(* move CaseData *)
IF fbExecute.Q = TRUE THEN

	(* shift data *)
	MEMMOVE(ADR(aFailedCACData[2]), ADR(aFailedCACData[1]), SIZEOF(aFailedCACData) - SIZEOF(aFailedCACData[1]));
	(* clear data *)
	MEMSET(ADR(aFailedCACData[1]), 16#00, SIZEOF(aFailedCACData[1]));

	IF stPrintCACData.ProductionTime ='' THEN
		stPrintCACData.ProductionDate := F_StringWildcard('#YYYYMMDD#', stCTDateTime.sSystemTime);
		stPrintCACData.ProductionTime := F_StringWildcard('#hhmmss#', stCTDateTime.sSystemTime);
		stPrintCACData.ProductionTimeOffset := F_SYSTEM_SystemTimeOffsetToHHMM(stCTDateTime.nSystemTimeOffset);
	END_IF

	MEMMOVE(ADR(aFailedCACData[1]), ADR(stPrintCACData), SIZEOF(aFailedCACData[1]));

	(*shift HMI Data*)
	MEMMOVE(ADR(aFailedCACDataHMI[2]), ADR(aFailedCACDataHMI[1]), SIZEOF(aFailedCACDataHMI) - SIZEOF(aFailedCACDataHMI[1]));
	(* clear data *)
	MEMSET(ADR(aFailedCACDataHMI[1]), 16#00, SIZEOF(aFailedCACDataHMI[1]));

	IF aFailedCACData[1].CaseRejectCode = 'OK' THEN
		aFailedCACDataHMI[1].sBarcode:= F_CONCAT3(aFailedCACData[1].Barcode,'(999)','1');
	ELSE
		aFailedCACDataHMI[1].sBarcode:= F_CONCAT3(aFailedCACData[1].Barcode,'(999)','0');
	END_IF

	(*IF aFailedCACData[1].Barcode <>  cCASE_PACKER_REJECT THEN
		aFailedCACDataHMI[1].sCaseIDCode		:= RIGHT(F_CODE_GetItem(aFailedCACData[1].Barcode, eCodeAIType.SerialCode, stCodeInfo_Case), 7);
	ELSE
		aFailedCACDataHMI[1].sCaseIDCode := '';
	END_IF
	aFailedCACDataHMI[1].sProductionDate 	:= aFailedCACData[1].ProductionDate;
	aFailedCACDataHMI[1].sProductionTime 	:= aFailedCACData[1].ProductionTime;
	aFailedCACDataHMI[1].sCaseRejectCode 	:= aFailedCACData[1].CaseRejectCode;*)
	aFailedCACDataHMI[1].nNumberOfOuters	:= aFailedCACData[1].NumberOfOuters;
	aFailedCACDataHMI[1].nNumberOfPacks 	:= aFailedCACData[1].Outer[1].NumberOfPacks;


	FOR nIndexOuter:=1 TO MIN(aFailedCACData[1].NumberOfOuters,cMAX_OUTERS_PER_CASE) DO
		IF aFailedCACData[1].Outer[nIndexOuter].OuterRejectCode = 'OK' THEN
			aFailedCACDataHMI[1].aOuter[nIndexOuter].sBarcode:= F_CONCAT3(aFailedCACData[1].Outer[nIndexOuter].Barcode,'(999)','1');
		ELSE
			aFailedCACDataHMI[1].aOuter[nIndexOuter].sBarcode:= F_CONCAT3(aFailedCACData[1].Outer[nIndexOuter].Barcode,'(999)','0');
		END_IF

		FOR nIndexPack:=1 TO MIN(aFailedCACData[1].Outer[nIndexOuter].NumberOfPacks, cMAX_PACKS_PER_OUTER) DO
			IF aFailedCACData[1].Outer[nIndexOuter].PackRejectCode[nIndexPack] = 'OK' THEN
				aFailedCACDataHMI[1].aOuter[nIndexOuter].aPackCode[nIndexPack]:= F_CONCAT3(aFailedCACData[1].Outer[nIndexOuter].PackCode[nIndexPack],'(999)','1');
			ELSE
				aFailedCACDataHMI[1].aOuter[nIndexOuter].aPackCode[nIndexPack]:= F_CONCAT3(aFailedCACData[1].Outer[nIndexOuter].PackCode[nIndexPack],'(999)','0');
			END_IF

		END_FOR
	END_FOR

	MEMSET(ADR(stQaseQueueDataHMI), 16#00, SIZEOF(stQaseQueueDataHMI));

	(*End of New HMI Data*)

	bDone := TRUE;

(* bExecute has been reset *)
ELSIF bExecute = FALSE THEN
	bDone := FALSE;
END_IF

END_FUNCTION_BLOCK

// ---- POUs/METS/Common LIB/04_CASE LIB/Case FBs/FB_CASE_MoveOutersRowToPacker.TcPOU
(* move Outers up to and including strOuterBarcode from sInfeedQueue to stCACData *)
FUNCTION_BLOCK FB_CASE_MoveOutersRowToPacker
VAR_INPUT
	bExecute 						: BOOL;		(* set TRUE to move Outers *)
	nOutersPerRow				: INT;
	nOutersPerCase				: INT;
	nPacker1Index					: INT;
	strOuterBarcode				: T_OUTER_Barcode;	(* 2D barcode from scanner *)
	sMetsSearchCode				: STRING(50); (*this is what to search for when changing the reject reason for FSS*)
	bUseInterimCodeForLastPosition	: BOOL;
	nAggregationQueueIndex			: INT;
	bManualConfirmationEnable		: BOOL;
END_VAR
VAR_IN_OUT
	sInfeedQueue				: ST_CASE_InfeedQueue;	(* Infeed Queue *)
	sPackerQueue 				: ST_CASE_InfeedQueue;	(* Outfeed Queue *)
	stCaseQueue				: ST_CASE_CaseQueue;				(* Outfeed Case Queue *)
	nRestoreCounter			: UDINT;
	stCodeInfo					: ST_CodeInfo;
END_VAR
VAR_OUTPUT
	bDone 					: BOOL;		(* TRUE = complete *)
	bBusy					: BOOL;		(* TRUE = in progress *)
	bError					: BOOL;		(* TRUE = error *)
	nErrorID					: UDINT;	(* error code *)
	nValidationIndex			: INT;
	bValIndexNotFound			: BOOL;
	sOutersMoved				: T_LongSTRING;
END_VAR
VAR
	fbExecute					: R_TRIG;
	eState					: E_CASE_State;
	eErrorState				: E_CASE_State;
	nOuterIndex				: T_PositiveINT;
	//nMaxInfeedIndex			: T_PositiveINT;
	nCaseQueueIndex			: T_PositiveINT;
	//nMaxCaseQueueIndex		: T_PositiveINT;
	nVALIndex					: INT;
	nRowIndex					: INT;
	sAppendedString				: STRING;
	(*nMaxOutersPerCase			: INT;*)
	nCounterDeletedLable		: INT;
	nQtyOver					: INT;
	nDeletedFiles				: UDINT;
	sDeletedBarcode			: T_OUTER_Barcode;	(* 2D barcode from scanner *)
	nMemoQtyOver			: INT;

	nValQtyOver				: INT;
END_VAR

(* rising edge of bExecute *)
fbExecute(CLK:= bExecute);

CASE eState OF

	(* idle *)
	E_CASE_IDLE:

		(* move Outers from sInfeedQueue to stCACData *)
		IF fbExecute.Q THEN

			(* update outputs *)
			bDone := FALSE;
			bBusy := TRUE;
			bError := FALSE;
			nErrorID := 0;
			eErrorState := eState;
			bValIndexNotFound := FALSE;

			sAppendedString	:= '';
			sOutersMoved 	:= '';
			
			(* max no of Outers in sInfeedQueue and sPackerQueue *)
			//nMaxInfeedIndex := TO_INT(SIZEOF(sInfeedQueue.aOuter) / SIZEOF(sInfeedQueue.aOuter[1]));

			(* reset nValidationIndex and get expected Outer barcode *)
			nValidationIndex := 0;
			nDeletedFiles := 0;
			(*
			(* clear and initialise stCACData *)
			MEMSET(ADR(stCACData), 16#00, SIZEOF(stCACData));*)

			eState := E_CASE_SCANINFEEDQUEUE;

		(* bExecute has been reset *)
		ELSIF bExecute = FALSE THEN

			(* update outputs *)
			bDone := FALSE;
			bBusy := FALSE;
			bError := FALSE;
			nErrorID := 0;
			bValIndexNotFound :=FALSE;
		END_IF


	(* find strOuterBarcode in sInfeedQueue *)
	E_CASE_SCANINFEEDQUEUE:

		IF strOuterBarcode <> '' THEN
			(* scan sInfeedQueue *)
			FOR nOuterIndex := 1 TO MIN(sInfeedQueue.nIndex, cMAX_INFEED_QUEUE)  DO
				(* strOuterBarcode found *)
				IF bManualConfirmationEnable THEN
					IF   sInfeedQueue.aOuter[nOuterIndex].Barcode = strOuterBarcode THEN

						nValidationIndex := sInfeedQueue.nIndex;
						EXIT;
					END_IF
				ELSIF (bUseInterimCodeForLastPosition AND sInfeedQueue.aOuter[nOuterIndex].AggregationCodes[1] = strOuterBarcode) OR
					(NOT bUseInterimCodeForLastPosition AND sInfeedQueue.aOuter[nOuterIndex].Barcode = strOuterBarcode)   THEN

					nValidationIndex := nOuterIndex - nAggregationQueueIndex;
					EXIT;
				END_IF
			END_FOR

			(* strOuterBarcode was found *)
			IF nValidationIndex > 0 AND nValidationIndex=nOutersPerRow*2 AND sPackerQueue.nIndex = 0  AND nPacker1Index = 0 THEN

				(* max no of Cases  in stCaseQueue *)
				//nMaxCaseQueueIndex := UDINT_TO_INT(SIZEOF(stCaseQueue.aCACData) / SIZEOF(stCaseQueue.aCACData[1]));
				(* scan stCaseQueue *)
				FOR nCaseQueueIndex := 1 TO cMAX_CASE_QUEUE DO

					(* strOuterBarcode found *)
					IF stCaseQueue.aCACData[nCaseQueueIndex].CaseRejectCode <> '' THEN

						IF FIND(stCaseQueue.aCACData[nCaseQueueIndex].CaseRejectCode, sMetsSearchCode) > 0 THEN
							nVALIndex := STRING_TO_INT(MID(stCaseQueue.aCACData[nCaseQueueIndex].CaseRejectCode ,2,7));
						ELSE
							nVALIndex := -1;
						END_IF

						IF nOutersPerCase = nVALIndex + nOutersPerRow AND nVALIndex > 0 AND nOutersPerCase > 0 AND nOutersPerRow > 0 THEN

							MEMMOVE(ADR(stCaseQueue.aCACData[nCaseQueueIndex].Outer[nVALIndex+1]), ADR(sInfeedQueue.aOuter[1]), F_SafeTo_UDINT(nOutersPerRow)* SIZEOF(sInfeedQueue.aOuter[1]));
							
							IF  nOutersPerRow = cMAX_INFEED_QUEUE THEN
								MEMSET(ADR(sInfeedQueue.aOuter), 16#00, SIZEOF(sInfeedQueue.aOuter));
							ELSIF nOutersPerRow < cMAX_INFEED_QUEUE THEN
								MEMMOVE(ADR(sInfeedQueue.aOuter[1]), ADR(sInfeedQueue.aOuter[nOutersPerRow + 1]), F_SafeTo_UDINT(cMAX_INFEED_QUEUE - nOutersPerRow) * SIZEOF(sInfeedQueue.aOuter[1]));
							END_IF
							
							sInfeedQueue.nIndex := LIMIT(0,sInfeedQueue.nIndex - nOutersPerRow,cMAX_INFEED_QUEUE);
							nValidationIndex :=nOutersPerRow - nAggregationQueueIndex;
							stCaseQueue.aCACData[nCaseQueueIndex]. NumberOfOuters := nOutersPerCase;
							stCaseQueue.aCACData[nCaseQueueIndex].CaseRejectCode := 'OK';
							stCaseQueue.aCACData[nCaseQueueIndex].CaseRejectID := 0;
						END_IF

						EXIT;
					END_IF
				END_FOR

				eState := E_CASE_UPDATEINFEEDQUEUE;

			ELSIF nValidationIndex > 0 THEN

				eState := E_CASE_UPDATEINFEEDQUEUE;

			(* strOuterBarcode not found *)
			ELSE

				bValIndexNotFound  := TRUE;

				(* update outputs *)
				bError := TRUE;
				nErrorID := 12;
				eErrorState := eState;

				sOutersMoved	:= F_CONCAT3('RowComplete moved [0]:', ' ErrorID: ', UDINT_TO_STRING(nErrorID));

				IF bManualConfirmationEnable THEN
					MEMSET(ADR(sInfeedQueue), 16#00, SIZEOF(sInfeedQueue));
				END_IF

				eState := E_CASE_DONE;
			END_IF

		(* strOuterBarcode does not contain data *)
		ELSE

			(* update outputs *)
			bError := TRUE;
			nErrorID := 11;
			eErrorState := eState;

			sOutersMoved	:= F_CONCAT3('RowComplete moved [0]:', ' ErrorID: ', UDINT_TO_STRING(nErrorID));

			eState := E_CASE_DONE;
		END_IF


	(* move Outers from sInfeedQueue to stCACData *)
	E_CASE_UPDATEINFEEDQUEUE:

		nQtyOver := nValidationIndex MOD nOutersPerRow;

		IF  nQtyOver <> 0 AND nValidationIndex <= cMAX_INFEED_QUEUE  THEN
			FOR nOuterIndex := 1 TO nValidationIndex DO
				IF sInfeedQueue.aOuter[nOuterIndex].OuterMasterListRestored  THEN

					sDeletedBarcode := sInfeedQueue.aOuter[nOuterIndex].Barcode;
					nMemoQtyOver := nQtyOver;

					IF nOuterIndex = cMAX_INFEED_QUEUE THEN
						MEMSET(ADR(sInfeedQueue.aOuter[cMAX_INFEED_QUEUE]), 16#00, SIZEOF(sInfeedQueue.aOuter[1]));
					ELSIF nOuterIndex < cMAX_INFEED_QUEUE THEN
						MEMMOVE(ADR(sInfeedQueue.aOuter[nOuterIndex]), ADR(sInfeedQueue.aOuter[nOuterIndex+1]), SIZEOF(sInfeedQueue.aOuter[1]) * F_SafeTo_UDINT(sInfeedQueue.nIndex - nOuterIndex) );
						MEMSET(ADR(sInfeedQueue.aOuter[sInfeedQueue.nIndex]), 16#00, SIZEOF(sInfeedQueue.aOuter[1]));
					END_IF
					
					nValidationIndex := nValidationIndex - 1;
					sInfeedQueue.nIndex := sInfeedQueue.nIndex - 1;

					nRestoreCounter	:= MAX(0, nRestoreCounter - 1);
					nDeletedFiles := nDeletedFiles + 1;
					nCounterDeletedLable :=nCounterDeletedLable + 1;
				END_IF
			END_FOR
		END_IF

		nValQtyOver := nValidationIndex MOD nOutersPerRow;

		IF  nValQtyOver <> 0  THEN
			FOR nOuterIndex := 1 TO nValidationIndex DO
				sInfeedQueue.aOuter[nOuterIndex].OuterCodeStatus.5 := TRUE;
			END_FOR
		END_IF

		(* move Outers from sInfeedQueue to sPackerQueue, clamped to max number of Outers supported by sPackerQueue *)
		IF cMAX_INFEED_QUEUE -  sPackerQueue.nIndex >= MIN(nValidationIndex, cMAX_INFEED_QUEUE) THEN
			MEMMOVE(ADR(sPackerQueue.aOuter[sPackerQueue.nIndex+1]), ADR(sInfeedQueue.aOuter[1]), F_SafeTo_UDINT(MIN(nValidationIndex, cMAX_INFEED_QUEUE)) * SIZEOF(sInfeedQueue.aOuter[1]));
		ELSIF cMAX_INFEED_QUEUE -  sPackerQueue.nIndex > 0 THEN
			MEMMOVE(ADR(sPackerQueue.aOuter[sPackerQueue.nIndex+1]), ADR(sInfeedQueue.aOuter[1]), F_SafeTo_UDINT(cMAX_INFEED_QUEUE - sPackerQueue.nIndex) * SIZEOF(sInfeedQueue.aOuter[1]));
		END_IF
		sPackerQueue.nIndex := LIMIT(0, sPackerQueue.nIndex + MIN(nValidationIndex, cMAX_INFEED_QUEUE),cMAX_INFEED_QUEUE);

		sOutersMoved	:= F_CONCAT3('RowComplete moved [', INT_TO_STRING(nValidationIndex), ']:');
		FOR nRowIndex :=1 TO nValidationIndex DO
			//sOutersMoved :=F_LongCONCAT(sOutersMoved, '   ');
			//sOutersMoved :=F_LongCONCAT(sOutersMoved, F_CODE_GetItem(sInfeedQueue.aOuter[nRowIndex].Barcode, eCodeAIType.SerialCode, stCodeInfo));
			
			CONCAT2(ADR(sOutersMoved), ADR('   '), ADR(sOutersMoved), SIZEOF(sOutersMoved));
		
			sAppendedString := RIGHT(F_CODE_GetItem(sInfeedQueue.aOuter[nRowIndex].Barcode, eCodeAIType.SerialCode, stCodeInfo),7);
			CONCAT2(ADR(sOutersMoved), ADR(sAppendedString), ADR(sOutersMoved), SIZEOF(sOutersMoved));
		END_FOR

		(* move remaining Outers forward in sInfeedQueue and update index pointer *)
		IF cMAX_INFEED_QUEUE - nValidationIndex > 0 THEN
			MEMMOVE(ADR(sInfeedQueue.aOuter[1]), ADR(sInfeedQueue.aOuter[nValidationIndex + 1]), F_SafeTo_UDINT(cMAX_INFEED_QUEUE - nValidationIndex) * SIZEOF(sInfeedQueue.aOuter[1]));
			sInfeedQueue.nIndex := LIMIT(0,sInfeedQueue.nIndex - nValidationIndex,cMAX_INFEED_QUEUE);
		END_IF

		(* clear all data for empty Outers in sInfeedQueue *)
		IF cMAX_INFEED_QUEUE - sInfeedQueue.nIndex > 0 THEN
			MEMSET(ADR(sInfeedQueue.aOuter[sInfeedQueue.nIndex + 1]), 16#00, F_SafeTo_UDINT(cMAX_INFEED_QUEUE - sInfeedQueue.nIndex ) * SIZEOF(sInfeedQueue.aOuter[1]));
		END_IF

		IF sInfeedQueue.bDoorReject THEN
			sPackerQueue.bDoorReject := TRUE;
			sInfeedQueue.bDoorReject := FALSE;
		END_IF

		eState := E_CASE_DONE;


	(* complete *)
	E_CASE_DONE:

		(* update outputs *)
		bDone := TRUE;
		bBusy := FALSE;

		eState := E_CASE_IDLE;


(* unknown state *)
ELSE

	eState := E_CASE_IDLE;

	(* clear outputs *)
	bDone := FALSE;
	bBusy := FALSE;
	bError := FALSE;
	nErrorID := 0;
END_CASE

END_FUNCTION_BLOCK

// ---- POUs/METS/Common LIB/04_CASE LIB/Case FBs/FB_CASE_MoveVerifiedCAC.TcPOU
(* move verified CaC data into table structure *)
FUNCTION_BLOCK FB_CASE_MoveVerifiedCAC
VAR_INPUT
	bExecute 						: BOOL;
	stPrintCACData				: ST_CAC_Data;
	stCTDateTime					: ST_SYSTEM_DateTime;
	(*stCodeInfo_Case				: ST_CodeInfo;*)
END_VAR
VAR_IN_OUT
	aVerifiedCACData				: ARRAY[1..cMAX_VERIFIED_CASE_QUEUE] OF ST_CAC_Data; 	(* array of verified CAC data *)
	aVerifiedCACDataHMI			: ARRAY[1..cMAX_VERIFIED_CASE_QUEUE] OF ST_HMI_CAC_Data; 	(* array of verified CAC data *)
	stQaseQueueDataHMI			: ST_HMI_CAC_Data;
END_VAR
VAR_OUTPUT
	bDone: BOOL;
END_VAR
VAR
	fbExecute						: R_TRIG;
	nIndexOuter					:INT;
	nIndexPack					:INT;
END_VAR

(* rising edge of bExecute *)
fbExecute(CLK:= bExecute);

(* move CaseData *)
IF fbExecute.Q = TRUE THEN

	(*shift data*)
	MEMMOVE(ADR(aVerifiedCACData[2]), ADR(aVerifiedCACData[1]), SIZEOF(aVerifiedCACData) - SIZEOF(aVerifiedCACData[1]));
	(* clear data *)
	MEMSET(ADR(aVerifiedCACData[1]), 16#00, SIZEOF(aVerifiedCACData[1]));

	IF stPrintCACData.ProductionTime ='' THEN
		stPrintCACData.ProductionDate := F_StringWildcard('#YYYYMMDD#', stCTDateTime.sSystemTime);
		stPrintCACData.ProductionTime := F_StringWildcard('#hhmmss#', stCTDateTime.sSystemTime);
		stPrintCACData.ProductionTimeOffset := F_SYSTEM_SystemTimeOffsetToHHMM(stCTDateTime.nSystemTimeOffset);
	END_IF

	MEMMOVE(ADR(aVerifiedCACData[1]), ADR(stPrintCACData), SIZEOF(aVerifiedCACData[1]));

	(*shift HMI Data*)
	MEMMOVE(ADR(aVerifiedCACDataHMI[2]), ADR(aVerifiedCACDataHMI[1]), SIZEOF(aVerifiedCACDataHMI) - SIZEOF(aVerifiedCACDataHMI[1]));
	(* clear data *)
	MEMSET(ADR(aVerifiedCACDataHMI[1]), 16#00, SIZEOF(aVerifiedCACDataHMI[1]));

	IF aVerifiedCACData[1].CaseRejectCode = 'OK' THEN
		aVerifiedCACDataHMI[1].sBarcode:= F_CONCAT3(aVerifiedCACData[1].Barcode,'(999)','1');
	ELSE
		aVerifiedCACDataHMI[1].sBarcode:= F_CONCAT3(aVerifiedCACData[1].Barcode,'(999)','0');
	END_IF

	(*aVerifiedCACDataHMI[1].sCaseIDCode		:= RIGHT( F_CODE_GetItem(aVerifiedCACData[1].Barcode, eCodeAIType.SerialCode, stCodeInfo_Case), 7);
	aVerifiedCACDataHMI[1].sProductionDate 	:= aVerifiedCACData[1].ProductionDate;
	aVerifiedCACDataHMI[1].sProductionTime 	:= aVerifiedCACData[1].ProductionTime;
	aVerifiedCACDataHMI[1].sCaseRejectCode 	:= aVerifiedCACData[1].CaseRejectCode;*)
	aVerifiedCACDataHMI[1].nNumberOfOuters 	:= aVerifiedCACData[1].NumberOfOuters;
	aVerifiedCACDataHMI[1].nNumberOfPacks 	:= aVerifiedCACData[1].Outer[1].NumberOfPacks;



	FOR nIndexOuter:=1 TO MIN(aVerifiedCACData[1].NumberOfOuters,cMAX_OUTERS_PER_CASE) DO
		IF aVerifiedCACData[1].Outer[nIndexOuter].OuterRejectCode = 'OK' THEN
			aVerifiedCACDataHMI[1].aOuter[nIndexOuter].sBarcode:= F_CONCAT3(aVerifiedCACData[1].Outer[nIndexOuter].Barcode,'(999)','1');
		ELSE
			aVerifiedCACDataHMI[1].aOuter[nIndexOuter].sBarcode:= F_CONCAT3(aVerifiedCACData[1].Outer[nIndexOuter].Barcode,'(999)','0');
		END_IF

		FOR nIndexPack:=1 TO MIN(aVerifiedCACData[1].Outer[nIndexOuter].NumberOfPacks, cMAX_PACKS_PER_OUTER) DO
			IF aVerifiedCACData[1].Outer[nIndexOuter].PackRejectCode[nIndexPack] = 'OK' THEN
				aVerifiedCACDataHMI[1].aOuter[nIndexOuter].aPackCode[nIndexPack]:= F_CONCAT3(aVerifiedCACData[1].Outer[nIndexOuter].PackCode[nIndexPack],'(999)','1');
			ELSE
				aVerifiedCACDataHMI[1].aOuter[nIndexOuter].aPackCode[nIndexPack]:= F_CONCAT3(aVerifiedCACData[1].Outer[nIndexOuter].PackCode[nIndexPack],'(999)','0');
			END_IF

		END_FOR
	END_FOR

	MEMSET(ADR(stQaseQueueDataHMI), 16#00, SIZEOF(stQaseQueueDataHMI));

	(*End of New HMI Part*)

	bDone := TRUE;

(* bExecute has been reset *)
ELSIF bExecute = FALSE THEN
	bDone := FALSE;
END_IF

END_FUNCTION_BLOCK

// ---- POUs/METS/Common LIB/04_CASE LIB/Case FBs/FB_CASE_RestoreDataControl.TcPOU
FUNCTION_BLOCK FB_CASE_RestoreDataControl
VAR_INPUT
	bEnableRestoreOCV		: BOOL;
END_VAR
VAR_IN_OUT
	stInfeedQueue			: ST_CASE_InfeedQueue;
	aOuterStatus			: ARRAY[1..cMAX_OUTER_STATUS_QUEUE] OF ST_OUTER_Status;
	stProductInstruction		: ST_PCM_Status;
END_VAR
VAR_OUTPUT
	sLastCode			: T_OUTER_Barcode;
END_VAR
VAR
	nConvQueueIndex		: INT;
	nOuterIndex			: INT;
END_VAR


IF bEnableRestoreOCV  AND stProductInstruction.nOpMode = 11  THEN

	FOR nConvQueueIndex := 1 TO  MIN(stInfeedQueue.nIndex, cMAX_INFEED_QUEUE) DO
		IF stInfeedQueue.aOuter[nConvQueueIndex].Barcode <> '' AND stInfeedQueue.aOuter[nConvQueueIndex].NumberOfLinkedPacks = 0 THEN
			FOR nOuterIndex := 1 TO cMAX_OUTER_STATUS_QUEUE  DO
				IF aOuterStatus[nOuterIndex].stOACData.Barcode = stInfeedQueue.aOuter[nConvQueueIndex].Barcode 		AND
						aOuterStatus[nOuterIndex].nStatus.17 = TRUE 											AND
						(aOuterStatus[nOuterIndex].nStatus.10 = TRUE  OR aOuterStatus[nOuterIndex].nStatus.11 = TRUE ) 	THEN

					stInfeedQueue.aOuter[nConvQueueIndex] := aOuterStatus[nOuterIndex].stOACData;
					sLastCode := stInfeedQueue.aOuter[nConvQueueIndex].Barcode ;
				END_IF
			END_FOR
		END_IF
	END_FOR
END_IF

END_FUNCTION_BLOCK

// ---- POUs/METS/Common LIB/04_CASE LIB/Case FBs/FB_CASE_ShiftCaseQueue.TcPOU
(* shifts specified group of cases in CaseQueue by 1 index *)
FUNCTION_BLOCK FB_CASE_ShiftCaseQueue
VAR_INPUT
	bExecute					: BOOL;			(* set TRUE to shift Case Queue *)
	bLogCaseOwerwriten		: BOOL;
	stCTDateTime				: ST_SYSTEM_DateTime;
	nFirstCaseIndex			: INT;			(* index of 1st case to be shifted *)
	nLastCaseIndex			: INT;			(* index of last case position owerwriten *)
	bStopOnOverWrittenData	: BOOL;
	tTimeOut					: TIME;
END_VAR
VAR_IN_OUT
	stCACDataDB				: ST_DB_CACDataCtrl;
	stCaseQueue				: ST_CASE_CaseQueue;	(* Case Queue *)
	stCaseQueueHMI			: ST_HMI_CASE_CaseQueue;	(* Case Queue *)
	(*bFoundNotEmptyTarget		: BOOL;*)
END_VAR
VAR_OUTPUT
	bDone					: BOOL;			(* TRUE = complete *)
	bBusy					: BOOL;
	bError					: BOOL;			(* TRUE = nFirstIndex and nLastCaseIndex not valid *)
	nErrorID					: UDINT;
	bCACDataLogInDB				: BOOL;
	bFoundNotEmptyTarget		: BOOL;
END_VAR
VAR
	fbExecute					: R_TRIG;
	//nMaxCaseIndex			: INT;

	eStep					: E_CASE_State;
	eErrorState				: E_CASE_State;

	tonTimeOut				: TON;
	rtTimeOutExec				: R_TRIG;

	sCACFile				: T_MaxString;
	stCACDataToLog					:  ST_CAC_Data;	(* array of CAC data *)
	nCaseQueueToShift				: INT;
	(*bLogOwerwritenDataToFileEx		: BOOL;
	fbLogOwerwritenCACData		: FB_CAC_WriteFile;*)

END_VAR

(***************************************TimeOut *******************************************)
(* monitor Busy timeout *)
tonTimeOut( IN:=eStep=E_CASE_OVERWIRTECAC, PT:=tTimeOut, Q=>);
(*	cTHREE_SECONDS						: TIME := T#3s;
	cFIVE_SECONDS						: TIME := t#5s;
	cTEN_SECONDS						: TIME := t#10s;*)

rtTimeOutExec(CLK:= tonTimeOut.Q);

IF rtTimeOutExec.Q THEN

	bError := TRUE;
	nErrorID := 100;
	eErrorState := eStep;

	MEMSET(ADR(stCACDataDB), 16#00, SIZEOF(stCACDataDB));

	eStep := E_CASE_DATAFINALISE;
END_IF


(***************************************Execution*******************************************)

(* rising edge of bExecute *)
fbExecute(CLK:= bExecute);


CASE eStep OF

	E_CASE_IDLE:
		(* move CaseData *)
		IF fbExecute.Q = TRUE THEN

			bDone := FALSE;
			bBusy := TRUE;
			bError := FALSE;
			nErrorID	:= 0;

			eErrorState	:=eStep;
			(* max index of Case Queue buffer *)
			//nMaxCaseIndex := UDINT_TO_INT(SIZEOF(stCaseQueue.aCACData) / SIZEOF(stCaseQueue.aCACData[1]));
			bFoundNotEmptyTarget := FALSE;
			bCACDataLogInDB	:= FALSE;
			MEMSET(ADR(stCACDataToLog), 16#00, SIZEOF(stCACDataToLog));
			(*nLastCaseIndex := nFirstCaseIndex + nTotalCasesToShift ;*)
			eStep :=E_CASE_DATAVALIDATE;
	
		(* bExecute has been reset *)
		ELSIF bExecute = FALSE THEN
	
			bDone := FALSE;
			bBusy := FALSE;
			bError := FALSE;
			nErrorID	:= 0;

			bFoundNotEmptyTarget := FALSE;
	
		END_IF

	E_CASE_DATAVALIDATE:
		(* specified range within buffer limits *)
		IF nFirstCaseIndex > 0 AND nLastCaseIndex <= cMAX_CASE_QUEUE THEN

			nCaseQueueToShift := nLastCaseIndex-nFirstCaseIndex;
			(* cases to be shifted > 0 *)
			IF  nCaseQueueToShift > 0 THEN

				stCACDataToLog	:= stCaseQueue.aCACData[MAX(1, nLastCaseIndex)];

				eStep :=E_CASE_OVERWIRTECAC;

			ELSE
				bError := TRUE;
				eErrorState	:=eStep;
				nErrorID	:= 1;

				eStep :=E_CASE_DONE;
			END_IF
		(* nFirstIndex = 0 or specified range exceeds stCaseQueue limits *)
		ELSE
			bError := TRUE;
			eErrorState	:=eStep;
			nErrorID	:= 11;

			eStep :=E_CASE_DONE;
		END_IF

	E_CASE_OVERWIRTECAC:

		IF stCaseQueue.aCACData[nLastCaseIndex].CodingAndTrackingMode <> 0 AND bLogCaseOwerwriten THEN

			bFoundNotEmptyTarget := bStopOnOverWrittenData;

			IF F_InvalidateASCIIChar(F_CONCAT4('OVERWRITEN_Pos_',INT_TO_STRING(nLastCaseIndex),'_', F_SYSTEM_SystemTimeToCHM_Header(stCTDateTime.sSystemTime))) >	0 	THEN
	
				stCACDataDB.sFileCodeName	:= '';
			ELSE
				stCACDataDB.sFileCodeName	:= F_CONCAT4('OVERWRITEN_Pos_',INT_TO_STRING(nLastCaseIndex),'_', F_SYSTEM_SystemTimeToCHM_Header(stCTDateTime.sSystemTime));
			END_IF

			stCACDataDB.stCACStatusDB	:= stCACDataToLog;
			stCACDataDB.bBlockRecord	:= TRUE;
			stCACDataDB.bCreateDataReq	:= TRUE;

(*place for HectorDB block*)

			IF	stCACDataDB.bDone	THEN
		
				IF NOT  stCACDataDB.bError THEN
					bCACDataLogInDB	:= TRUE;
					sCACFile	:= stCACDataDB.sFileCodeName;
		
				ELSE
		
					bError := TRUE;
					nErrorID := stCACDataDB.nErrorID;
					eErrorState := eStep;
				END_IF

				eStep :=E_CASE_DATAFINALISE;
		
				MEMSET(ADR(stCACDataDB), 16#00, SIZEOF(stCACDataDB));
			END_IF
		ELSE
			eStep :=E_CASE_DATAFINALISE;
		END_IF

	E_CASE_DATAFINALISE:

		(* shift specified cases in CaseQueue *)
		MEMMOVE(ADR(stCaseQueue.aCACData[nFirstCaseIndex + 1]), ADR(stCaseQueue.aCACData[nFirstCaseIndex]), F_SafeTo_UDINT(nCaseQueueToShift)* SIZEOF(stCaseQueue.aCACData[1]));

		(* shift specified cases in CaseQueue *)
		MEMMOVE(ADR(stCaseQueueHMI.aCACData[nFirstCaseIndex + 1]), ADR(stCaseQueueHMI.aCACData[nFirstCaseIndex]), F_SafeTo_UDINT(nCaseQueueToShift)* SIZEOF(stCaseQueueHMI.aCACData[1]));

		(* clear data in 1st indexes *)
		MEMSET(ADR(stCaseQueue.aCACData[nFirstCaseIndex]), 16#00, SIZEOF(stCaseQueue.aCACData[nFirstCaseIndex]));

		(* clear data in 1st indexes *)
		MEMSET(ADR(stCaseQueueHMI.aCACData[nFirstCaseIndex]), 16#00, SIZEOF(stCaseQueueHMI.aCACData[nFirstCaseIndex]));

		eStep :=E_CASE_DONE;

	E_CASE_DONE:

		bFoundNotEmptyTarget := FALSE;

		bDone := TRUE;
		bBusy := FALSE;

		eStep :=E_CASE_IDLE;
ELSE
	eStep :=E_CASE_IDLE;
END_CASE

END_FUNCTION_BLOCK

// ---- POUs/METS/Common LIB/04_CASE LIB/Case FBs/FB_CASE_ValidatePrintCACData.TcPOU
FUNCTION_BLOCK FB_CASE_ValidatePrintCACData
VAR_INPUT
	bExecute						: BOOL;			(* set TRUE to load stPrintCACData *)
	bResetAlarmBits				: BOOL;
	strLastBarcode					: T_CASE_Barcode;
	bEnableCheckForDuplicates	: BOOL;
	bEnableCaseContentReject		: BOOL;
	bEnableStopOnCaseInavlid		: BOOL;
	bCaseRejectedByCasePacker 		: BOOL;
	stCTDateTime					: ST_SYSTEM_DateTime;	(* CaseTrace date/time structure *)
	stCodeInfo_Case				: ST_CodeInfo;
END_VAR
VAR_IN_OUT
	stProductInstruction				: ST_PCM_Status; (* Product Instruction *)
	stCaseRejectReasons					: ST_RejectReasonsForCase;
	stFirstCACData					: ST_CAC_Data;	(* source CAC data for valid case *)
	stLastCACData						: ST_CAC_Data;	(* source CAC data for valid case *)
	stPrintCACData					: ST_CAC_Data;	(* CAC data to generate case label *)
	aLastCaseBarcodes				: ARRAY[1..cMAX_LAST_CASE_BARCODES] OF T_CASE_Barcode;
END_VAR
VAR_OUTPUT
	bDone						: BOOL;			(* TRUE = complete *)
	bDuplicateCaseLabelFound		: BOOL;
	bCaseLabelInvalidDataFound		: BOOL;
	bDoorGuardRejectFound			: BOOL;
	sDuplicatedLabel				: T_CASE_Barcode;
	nIndex						: INT;
END_VAR
VAR
	fbExecute						: R_TRIG;
	fbValidateCaseLabel				: FB_CODE_ValidateExplicitCode;
	strPreviousBarcode				: T_CASE_Barcode;
	nRejectIndex					: INT;

	nOuterIndex					: INT;
	nPackInex						: INT;

	bInvalidRejectCode					: BOOL;

	aStatusErrorVal					: ARRAY[0..10] OF STRING(10);
	aRejectCodePointer     		   	: ARRAY[0..10] OF STRING(10);

END_VAR

(* rising edge of bExecute *)
fbExecute(CLK:= bExecute);

IF bResetAlarmBits THEN
	bDuplicateCaseLabelFound := FALSE;
	bCaseLabelInvalidDataFound	:= FALSE;
END_IF

(* move CaseData *)
IF fbExecute.Q = TRUE THEN


	IF bCaseRejectedByCasePacker	AND bEnableCaseContentReject THEN
		(* copy CAC data from source to target *)
		MEMMOVE(ADR(stPrintCACData), ADR(stFirstCACData), SIZEOF(stFirstCACData));
		(* clear source CAC data *)
		MEMSET(ADR(stFirstCACData), 16#00, SIZEOF(stFirstCACData));
	ELSE
		(* copy CAC data from source to target *)
		MEMMOVE(ADR(stPrintCACData), ADR(stLastCACData), SIZEOF(stLastCACData));
		(* clear source CAC data *)
		MEMSET(ADR(stLastCACData), 16#00, SIZEOF(stLastCACData));
	END_IF

	(*Print barcode*)
	stPrintCACData.Barcode 		:=strLastBarcode;
	bDuplicateCaseLabelFound	:= FALSE;
	bCaseLabelInvalidDataFound	:= FALSE;
	bDoorGuardRejectFound		:= FALSE;
	bInvalidRejectCode 			:= FALSE;
	sDuplicatedLabel := '';

	(*IF stPrintCACData.ProductionTime ='' THEN*)
	stPrintCACData.ProductionDate := F_StringWildcard('#YYYYMMDD#', stCTDateTime.sSystemTime);
	stPrintCACData.ProductionTime := F_StringWildcard('#hhmmss#', stCTDateTime.sSystemTime);
	stPrintCACData.ProductionTimeOffset := F_SYSTEM_SystemTimeOffsetToHHMM(stCTDateTime.nSystemTimeOffset);
	(*END_IF*)

	IF NOT  stProductInstruction.bEnableAggregation THEN
		stPrintCACData.CaseRejectCode 	:= 'OK';
		stPrintCACData.CaseRejectID		:= 0;
	END_IF

	fbValidateCaseLabel(	sFullCode := stPrintCACData.Barcode,
								stCodeInfo := stCodeInfo_Case,
								stProductInstruction := stProductInstruction);

	IF stPrintCACData.CaseRejectCode = stCaseRejectReasons.stDoorGuardReject.sMetsDisplayCode THEN

(*------->check conseqences----------*)	(*stPrintCACData.Barcode := '';*)
			bDoorGuardRejectFound		:= TRUE;

	ELSIF  bCaseRejectedByCasePacker AND stPrintCACData.CaseRejectCode = 'OK' THEN

			stPrintCACData.CaseRejectCode := stCaseRejectReasons.stCasePackerReject.sMetsDisplayCode;
			stPrintCACData.CaseRejectID := stCaseRejectReasons.stCasePackerReject.nRejectID;

	ELSIF stProductInstruction.bEnableAggregation AND  fbValidateCaseLabel.bValidationOK AND stPrintCACData.Barcode = strPreviousBarcode THEN

			bDuplicateCaseLabelFound := TRUE;
			stPrintCACData.CaseRejectCode := stCaseRejectReasons.stCaseLabelDuplicate.sMetsDisplayCode;
			stPrintCACData.CaseRejectID := stCaseRejectReasons.stCaseLabelDuplicate.nRejectID;
			sDuplicatedLabel := stPrintCACData.Barcode;
	ELSE

		IF stPrintCACData.CaseRejectCode = 'OK' AND stPrintCACData.Barcode <> cCASE_PACKER_REJECT THEN

			IF stPrintCACData.Barcode = '' THEN
				stPrintCACData.CaseRejectCode := stCaseRejectReasons.stNoCaseLabelError.sMetsDisplayCode;
				stPrintCACData.CaseRejectID := stCaseRejectReasons.stNoCaseLabelError.nRejectID;
			ELSIF fbValidateCaseLabel.bEntireCodeLengthOK = FALSE THEN
				stPrintCACData.CaseRejectCode := stCaseRejectReasons.stCaseBarcodeInvalidLength.sMetsDisplayCode;
				stPrintCACData.CaseRejectID := stCaseRejectReasons.stCaseBarcodeInvalidLength.nRejectID;
			ELSIF fbValidateCaseLabel.bGtinOK = FALSE THEN
				stPrintCACData.CaseRejectCode := stCaseRejectReasons.stCaseLabelGtinError.sMetsDisplayCode;
				stPrintCACData.CaseRejectID := stCaseRejectReasons.stCaseLabelGtinError.nRejectID;
			ELSIF fbValidateCaseLabel.bBrandOK = FALSE THEN
				stPrintCACData.CaseRejectCode := stCaseRejectReasons.stCaseLabelBrandCodeError.sMetsDisplayCode;
				stPrintCACData.CaseRejectID := stCaseRejectReasons.stCaseLabelBrandCodeError.nRejectID;
			ELSIF fbValidateCaseLabel.bRskuOK = FALSE THEN
				stPrintCACData.CaseRejectCode := stCaseRejectReasons.stCaseLabelRskuError.sMetsDisplayCode;
				stPrintCACData.CaseRejectID := stCaseRejectReasons.stCaseLabelRskuError.nRejectID;
			ELSIF fbValidateCaseLabel.bProductionOrderOK = FALSE THEN
				stPrintCACData.CaseRejectCode := stCaseRejectReasons.stCaseLabelProductionOrderError.sMetsDisplayCode;
				stPrintCACData.CaseRejectID := stCaseRejectReasons.stCaseLabelProductionOrderError.nRejectID;
			ELSIF fbValidateCaseLabel.bBatchIDOK = FALSE THEN
				stPrintCACData.CaseRejectCode := stCaseRejectReasons.stCaseLabelBatchIDError.sMetsDisplayCode;
				stPrintCACData.CaseRejectID := stCaseRejectReasons.stCaseLabelBatchIDError.nRejectID;
			ELSIF fbValidateCaseLabel.bSerialCodeOK = FALSE THEN
				stPrintCACData.CaseRejectCode := stCaseRejectReasons.stCaseLabelSerialCodeError.sMetsDisplayCode;
				stPrintCACData.CaseRejectID := stCaseRejectReasons.stCaseLabelSerialCodeError.nRejectID;
			END_IF

			IF stPrintCACData.Barcode <> ''  AND NOT fbValidateCaseLabel.bValidationOK AND bEnableStopOnCaseInavlid THEN

				bCaseLabelInvalidDataFound := TRUE;

			ELSIF  stPrintCACData.Barcode <> '' AND bEnableCheckForDuplicates THEN

				(* Check for Duplicate Case Labeles in a Last Case Barcode Labels array *)
				FOR nIndex := 1 TO cMAX_LAST_CASE_BARCODES DO
					IF stPrintCACData.Barcode = aLastCaseBarcodes[nIndex] AND aLastCaseBarcodes[nIndex] <> '' AND aLastCaseBarcodes[nIndex] <> cCASE_PACKER_REJECT THEN
						bDuplicateCaseLabelFound := TRUE;
						stPrintCACData.CaseRejectCode := stCaseRejectReasons.stCaseLabelDuplicate.sMetsDisplayCode;
						stPrintCACData.CaseRejectID := stCaseRejectReasons.stCaseLabelDuplicate.nRejectID;
						sDuplicatedLabel := stPrintCACData.Barcode;
						EXIT;
					END_IF
				END_FOR
			END_IF

			IF stPrintCACData.CaseRejectCode = 'OK' THEN

				FOR nOuterIndex:= 1 TO MIN(stPrintCACData.NumberOfOuters, cMAX_OUTERS_PER_CASE) DO
					IF stPrintCACData.Outer[nOuterIndex].OuterRejectCode =  'OK' THEN
						FOR nPackInex :=1 TO MIN(stPrintCACData.Outer[nOuterIndex].NumberOfPacks, cMAX_PACKS_PER_OUTER) DO
							IF stPrintCACData.Outer[nOuterIndex].PackRejectCode[nPackInex] <> 'OK' THEN
								bInvalidRejectCode := TRUE;
								EXIT;
							END_IF
						END_FOR
					ELSE
						bInvalidRejectCode := TRUE;
					END_IF

					IF bInvalidRejectCode THEN
						aStatusErrorVal[0] 		:=  INT_TO_STRING(nOuterIndex);
						aRejectCodePointer[0] 	:= 'nn';

						stPrintCACData.CaseRejectCode 	:=	F_CODE_AssignValToStringWithPrefix(stCaseRejectReasons.stINVError.sMetsDisplayCode, aStatusErrorVal, aRejectCodePointer, 2, '0');
						stPrintCACData.CaseRejectID 		:= 	stCaseRejectReasons.stINVError.nRejectID;
						EXIT;
					END_IF
				END_FOR
			END_IF

		ELSIF stPrintCACData.CaseRejectCode = '' THEN

			stPrintCACData.CaseRejectCode :=stCaseRejectReasons.stCaseNoCaseData.sMetsDisplayCode;
			stPrintCACData.CaseRejectID :=stCaseRejectReasons.stCaseNoCaseData.nRejectID;
		END_IF
	END_IF

	(* update output *)
	strPreviousBarcode := stPrintCACData.Barcode;

	bDone := TRUE;

(* bExecute has been reset *)
ELSIF bExecute = FALSE THEN

	(* clear output *)
	bDone := FALSE;

END_IF

END_FUNCTION_BLOCK

// ---- POUs/METS/Common LIB/04_CASE LIB/Case Functons/F_CASE_AddAIBrackets.TcPOU
(* adds brackets around Application Identifiers (AI) in 1D barcode *)
FUNCTION F_CASE_AddAIBrackets : T_CASE_Barcode
VAR_INPUT
	strCaseBarcode		: T_CASE_Barcode;
END_VAR
VAR_IN_OUT
	stCodeInfo_Case		: ST_CodeInfo;
END_VAR
VAR
	strAI01				: T_MaxString;
	strAI10				: T_MaxString;
	strAI21				: T_MaxString;
	strAI91				: T_MaxString;
	strAI240				: T_MaxString;
	nNextPos: INT;
END_VAR

(* barcode does not contain any brackets *)
IF FIND(strCaseBarcode, '(') = 0 AND FIND(strCaseBarcode, ')') = 0 THEN


	(* break barcode into constituent parts *)
	IF	stCodeInfo_Case.stGTIN.nCodeLength <> 0 THEN
		strAI01 := LEFT(strCaseBarcode,  stCodeInfo_Case.stGTIN.nCodeLength + 2);
	END_IF

	IF	stCodeInfo_Case.stBatchID.nCodeLength  <> 0 THEN
		strAI10 := MID(strCaseBarcode, stCodeInfo_Case.stBatchID.nCodeLength + 2 , LEN(strAI01) + 1);
	END_IF

	IF	stCodeInfo_Case.stSerialCode.nCodeLength <> 0  THEN
		strAI21 := MID(strCaseBarcode, stCodeInfo_Case.stSerialCode.nCodeLength + 2 , LEN(strAI01) +  LEN(strAI10) + 1);
	END_IF

	nNextPos := LEN(strAI01)+ LEN(strAI10) + LEN(strAI21)+1;

	(* replace AI with AI in brackets *)
	IF	strAI01 <> '' THEN
		strAI01 := REPLACE(strAI01, '(01)', 2, 1);
	END_IF

	IF	strAI10 <> '' THEN
		strAI10 := REPLACE(strAI10, '(10)', 2, 1);
	END_IF

	IF	strAI21 <> ''  THEN
		strAI21 := REPLACE(strAI21, '(21)', 2, 1);
	END_IF

	(* 01MMMMMMMMMMMMMM240RRRRRRRR10SSSLLLDDDDHHMMSS *)
	IF MID(strCaseBarcode, 3, nNextPos) = '240' THEN
		IF	stCodeInfo_Case.stRSKU.nCodeLength  <> 0 THEN
			strAI240 := MID(strCaseBarcode, stCodeInfo_Case.stRSKU.nCodeLength + 3, nNextPos);
			nNextPos :=  nNextPos + LEN(strAI240);
			strAI240 := REPLACE(strAI240, '(240)', 3, 1);
		END_IF

		IF	stCodeInfo_Case.stProductionOrder.nCodeLength <> 0 THEN
			strAI91 := MID(strCaseBarcode, stCodeInfo_Case.stProductionOrder.nCodeLength + 2, nNextPos);
			strAI91 := REPLACE(strAI91, '(91)', 2, 1);
		END_IF

		F_CASE_AddAIBrackets := F_CONCAT5(strAI01, strAI10, strAI21, strAI240, strAI91);

	(* 01MMMMMMMMMMMMMM91RRRRRRRR10SSSLLLDDDDHHMMSS *)
	ELSE
		IF	stCodeInfo_Case.stProductionOrder.nCodeLength <> 0 THEN
			strAI91 := MID(strCaseBarcode, stCodeInfo_Case.stProductionOrder.nCodeLength + 2, nNextPos);
			nNextPos :=  nNextPos + LEN(strAI91);
			strAI91 := REPLACE(strAI91, '(91)', 2, 1);
		END_IF

		IF	stCodeInfo_Case.stRSKU.nCodeLength  <> 0 THEN
			strAI240 := MID(strCaseBarcode, stCodeInfo_Case.stRSKU.nCodeLength + 3, nNextPos);
			strAI240 := REPLACE(strAI240, '(240)', 3, 1);
		END_IF

		F_CASE_AddAIBrackets := F_CONCAT5(strAI01, strAI10, strAI21, strAI91, strAI240);
	END_IF

(* brackets already in barcode *)
ELSE

	F_CASE_AddAIBrackets := strCaseBarcode;
END_IF

END_FUNCTION

// ---- POUs/METS/Common LIB/04_CASE LIB/Case Functons/F_CASE_BarcodeToCACFilename.TcPOU
(* generates CAC filename from Case Barcode *)
FUNCTION F_CASE_BarcodeToCACFilename : T_CAC_Filename
VAR_INPUT
	sCaseBarcode					: T_CASE_Barcode;
	stDateTime					: TIMESTRUCT;
	bCaseRejectedByCasePacker	: BOOL;
END_VAR
(*VAR
	strDecryptedDate	: STRING(8);
END_VAR*)

sCaseBarcode	:= F_ReplaceSingleChar(sCaseBarcode, '\','');
sCaseBarcode	:= F_ReplaceSingleChar(sCaseBarcode, '/','');
sCaseBarcode	:= F_ReplaceSingleChar(sCaseBarcode, ':','');
sCaseBarcode	:= F_ReplaceSingleChar(sCaseBarcode, '*','');
sCaseBarcode	:= F_ReplaceSingleChar(sCaseBarcode, '?','');
sCaseBarcode	:= F_ReplaceSingleChar(sCaseBarcode, '<','');
sCaseBarcode	:= F_ReplaceSingleChar(sCaseBarcode, '>','');
sCaseBarcode	:= F_ReplaceSingleChar(sCaseBarcode, '|','');

IF sCaseBarcode <> '' AND NOT bCaseRejectedByCasePacker THEN
	F_CASE_BarcodeToCACFilename := F_SCANNER_RemoveAIBrackets(sCaseBarcode);
ELSIF bCaseRejectedByCasePacker THEN
	F_CASE_BarcodeToCACFilename := F_CONCAT3(sCaseBarcode,'_', F_SYSTEM_SystemTimeToCHM_Header(stDateTime));
ELSE
	F_CASE_BarcodeToCACFilename := CONCAT('NOCASELABEL_', F_SYSTEM_SystemTimeToCHM_Header(stDateTime));
END_IF

END_FUNCTION

// ---- POUs/METS/Common LIB/08_SOFTWARE LIB/String FBs/F_ReplaceSingleChar.TcPOU
FUNCTION F_ReplaceSingleChar : STRING(255)
VAR_INPUT
	sFullCode		: STRING(255);
	sCharRemove			: T_Char := '$1D';
	sReplacmentChar		: T_Char := '';
END_VAR
VAR
END_VAR

(* reset output *)
F_ReplaceSingleChar :='';

WHILE FIND(sFullCode, sCharRemove) > 0 DO
	sFullCode := REPLACE(sFullCode,sReplacmentChar, LEN(sCharRemove), FIND(sFullCode, sCharRemove));
END_WHILE

F_ReplaceSingleChar	:= sFullCode;

END_FUNCTION

// ---- POUs/METS/Common LIB/04_CASE LIB/Case Functons/F_CASE_ClearCACData.TcPOU
(* clear all data from Case Data *)
FUNCTION F_CASE_ClearCACData : BOOL
VAR_INPUT
	bEnable				: BOOL;			(* set TRUE to reset all values in Case Data *)
END_VAR

VAR_IN_OUT
	stCACData 			: ST_CAC_Data;	(* Case Data structure *)
END_VAR

(* clear stCACData enabled *)
IF bEnable = TRUE THEN

	(* reset stCACData *)
	MEMSET(ADR(stCACData), 16#00, SIZEOF(stCACData));

	(* set output to TRUE when reset is active *)
	F_CASE_ClearCACData := TRUE;

(* clear stCACData disabled *)
ELSE

	(* reset output *)
	F_CASE_ClearCACData := FALSE;
END_IF

END_FUNCTION

// ---- POUs/METS/Common LIB/04_CASE LIB/Case Functons/F_CASE_ClearCaseQueue.TcPOU
(* clear all data from Case Data *)
FUNCTION F_CASE_ClearCaseQueue : BOOL
VAR_INPUT
	bEnable				: BOOL;			(* set TRUE to reset all values in Case Data *)
END_VAR


VAR_IN_OUT
	stCaseQueue							: ST_CASE_CaseQueue;(* Case Data structure *)
	stCaseQueueHMI						:ST_HMI_CASE_CaseQueue;(* Case Data structure *)
END_VAR

(* clear stCaseQueue enabled *)
IF bEnable = TRUE THEN

	(* reset stCaseQueue *)
	MEMSET(ADR(stCaseQueue), 16#00, SIZEOF(stCaseQueue));

	(* reset aCaseQueueHMI *)
	MEMSET(ADR(stCaseQueueHMI), 16#00, SIZEOF(stCaseQueueHMI));

	(* set output to TRUE when reset is active *)
	F_CASE_ClearCaseQueue := TRUE;

(* clear stCaseQueue disabled *)
ELSE

	(* reset output *)
	F_CASE_ClearCaseQueue := FALSE;
END_IF

END_FUNCTION

// ---- POUs/METS/Common LIB/04_CASE LIB/Case Functons/F_CASE_ClearFailedCaseQueue.TcPOU
(* clear all data from Case Data *)
FUNCTION F_CASE_ClearFailedCaseQueue : BOOL
VAR_INPUT
	bEnable				: BOOL;			(* set TRUE to reset all values in Case Data *)
END_VAR

VAR_IN_OUT
	aFailedCACData						: ARRAY[1..cMAX_FAILED_CASE_QUEUE] OF ST_CAC_Data;
END_VAR

(* clear aFailedCACData enabled *)
IF bEnable = TRUE THEN

	(* reset aFailedCACData *)
	MEMSET(ADR(aFailedCACData), 16#00, SIZEOF(aFailedCACData));

	(* set output to TRUE when reset is active *)
	F_CASE_ClearFailedCaseQueue := TRUE;

(* clear aFailedCACData disabled *)
ELSE

	(* reset output *)
	F_CASE_ClearFailedCaseQueue := FALSE;
END_IF

END_FUNCTION

// ---- POUs/METS/Common LIB/04_CASE LIB/Case Functons/F_CASE_ClearInfeedQueue.TcPOU
(* clear all data from Case Data *)
FUNCTION F_CASE_ClearInfeedQueue : BOOL
VAR_INPUT
	bEnable				: BOOL;			(* set TRUE to reset all values in Case Data *)
END_VAR

VAR_IN_OUT
	stInfeedConvQueue 			: ST_CASE_InfeedQueue;	(* Case Data structure *)
END_VAR

(* clear stInfeedConvQueue enabled *)
IF bEnable = TRUE THEN

	(* reset stInfeedConvQueue *)
	MEMSET(ADR(stInfeedConvQueue), 16#00, SIZEOF(stInfeedConvQueue));

	(* set output to TRUE when reset is active *)
	F_CASE_ClearInfeedQueue := TRUE;

(* clear stInfeedConvQueue disabled *)
ELSE

	(* reset output *)
	F_CASE_ClearInfeedQueue := FALSE;
END_IF

END_FUNCTION

// ---- POUs/METS/Common LIB/04_CASE LIB/Case Functons/F_CASE_ClearPackerQueue.TcPOU
(* clear all data from Case Data *)
FUNCTION F_CASE_ClearPackerQueue : BOOL
VAR_INPUT
	bEnable				: BOOL;			(* set TRUE to reset all values in Case Data *)
END_VAR

VAR_IN_OUT
	aPackerQueue							: ARRAY [0..1] OF ST_CASE_InfeedQueue;	(* Case Data structure *)
END_VAR

(* clear aPackerQueue enabled *)
IF bEnable = TRUE THEN

	(* reset aPackerQueue *)
	MEMSET(ADR(aPackerQueue), 16#00, SIZEOF(aPackerQueue));

	(* set output to TRUE when reset is active *)
	F_CASE_ClearPackerQueue := TRUE;

(* clear aPackerQueue disabled *)
ELSE

	(* reset output *)
	F_CASE_ClearPackerQueue := FALSE;
END_IF

END_FUNCTION

// ---- POUs/METS/Common LIB/04_CASE LIB/Case Functons/F_CASE_GetRejectReasonFSS.TcPOU
FUNCTION F_CASE_GetRejectReasonFSS : T_FSS_RejecCode
VAR_INPUT
	sRejectReasonME			:	STRING(255);
	stCaseRejectReasons		: 	ST_RejectReasonsForCase;
END_VAR
VAR
	sRejectReasonFSS:	T_FSS_RejecCode;
END_VAR

IF sRejectReasonME = 'OK' THEN
	sRejectReasonFSS := '';

ELSIF sRejectReasonME = '' THEN
	sRejectReasonFSS := stCaseRejectReasons.stUnknownCaseReject.sFssSendCode;

ELSIF FIND(sRejectReasonME, stCaseRejectReasons.stValError.sMetsSearchCode) > 0 THEN
	sRejectReasonFSS := stCaseRejectReasons.stValError.sFssSendCode;

ELSIF FIND(sRejectReasonME, stCaseRejectReasons.stOACError.sMetsSearchCode) > 0 THEN
	sRejectReasonFSS := stCaseRejectReasons.stOACError.sFssSendCode;

ELSIF FIND(sRejectReasonME, stCaseRejectReasons.stINVError.sMetsSearchCode) > 0 THEN
	sRejectReasonFSS := stCaseRejectReasons.stINVError.sFssSendCode;

ELSIF FIND(sRejectReasonME, stCaseRejectReasons.stDUPError.sMetsSearchCode) > 0 THEN
	sRejectReasonFSS := stCaseRejectReasons.stDUPError.sFssSendCode;

ELSIF FIND(sRejectReasonME, stCaseRejectReasons.stPackNotLinedError.sMetsSearchCode) > 0 THEN
	sRejectReasonFSS := stCaseRejectReasons.stPackNotLinedError.sFssSendCode;

ELSIF FIND(sRejectReasonME, stCaseRejectReasons.stOuterGTINError.sMetsSearchCode) > 0 THEN
	sRejectReasonFSS := stCaseRejectReasons.stOuterGTINError.sFssSendCode;


ELSIF FIND(sRejectReasonME, stCaseRejectReasons.stOuterSerialError.sMetsSearchCode) > 0 THEN
	sRejectReasonFSS := stCaseRejectReasons.stOuterSerialError.sFssSendCode;

ELSIF FIND(sRejectReasonME, stCaseRejectReasons.stOuterRSKUError.sMetsSearchCode) > 0 THEN
	sRejectReasonFSS := stCaseRejectReasons.stOuterRSKUError.sFssSendCode;


ELSIF FIND(sRejectReasonME, stCaseRejectReasons.stNoCaseLabelError.sMetsSearchCode) > 0 THEN
	sRejectReasonFSS := stCaseRejectReasons.stNoCaseLabelError.sFssSendCode;

ELSIF FIND(sRejectReasonME, stCaseRejectReasons.stCasePackerReject.sMetsSearchCode) > 0 THEN
	sRejectReasonFSS := stCaseRejectReasons.stCasePackerReject.sFssSendCode;

ELSIF FIND(sRejectReasonME,stCaseRejectReasons.stDoorGuardReject.sMetsSearchCode) > 0 THEN
	sRejectReasonFSS := stCaseRejectReasons.stDoorGuardReject.sFssSendCode;

ELSIF FIND(sRejectReasonME, stCaseRejectReasons.stCaseLabelGtinError.sMetsSearchCode) > 0 THEN
	sRejectReasonFSS := stCaseRejectReasons.stCaseLabelGtinError.sFssSendCode;

ELSIF FIND(sRejectReasonME, stCaseRejectReasons.stCaseLabelProductionOrderError.sMetsSearchCode) > 0 THEN
	sRejectReasonFSS := stCaseRejectReasons.stCaseLabelProductionOrderError.sFssSendCode;

ELSIF FIND(sRejectReasonME, stCaseRejectReasons.stCaseLabelBatchIDError.sMetsSearchCode) > 0 THEN
	sRejectReasonFSS := stCaseRejectReasons.stCaseLabelBatchIDError.sFssSendCode;

ELSIF FIND(sRejectReasonME, stCaseRejectReasons.stCaseLabelRskuError.sMetsSearchCode) > 0 THEN
	sRejectReasonFSS := stCaseRejectReasons.stCaseLabelRskuError.sFssSendCode;

ELSIF FIND(sRejectReasonME, stCaseRejectReasons.stCaseLabelSerialCodeError.sMetsSearchCode) > 0 THEN
	sRejectReasonFSS := stCaseRejectReasons.stCaseLabelSerialCodeError.sFssSendCode;

ELSIF FIND(sRejectReasonME, stCaseRejectReasons.stCaseLabelDuplicate.sMetsSearchCode) > 0 THEN
	sRejectReasonFSS := stCaseRejectReasons.stCaseLabelDuplicate.sFssSendCode;

ELSIF FIND(sRejectReasonME, stCaseRejectReasons.stCaseNoCaseData.sMetsSearchCode) > 0 THEN
	sRejectReasonFSS := stCaseRejectReasons.stCaseNoCaseData.sFssSendCode;

ELSIF FIND(sRejectReasonME, stCaseRejectReasons.stCaseBarcodeInvalidLength.sMetsSearchCode) > 0 THEN
	sRejectReasonFSS := stCaseRejectReasons.stCaseBarcodeInvalidLength.sFssSendCode;

ELSIF FIND(sRejectReasonME, stCaseRejectReasons.stCaseDBInvalidCheck.sMetsSearchCode) > 0 THEN
	sRejectReasonFSS := stCaseRejectReasons.stCaseDBInvalidCheck.sFssSendCode;

ELSIF FIND(sRejectReasonME, stCaseRejectReasons.stCaseWhitelistInvalidCheck.sMetsSearchCode) > 0 THEN
	sRejectReasonFSS := stCaseRejectReasons.stCaseWhitelistInvalidCheck.sFssSendCode;

ELSIF FIND(sRejectReasonME, stCaseRejectReasons.stOuterBrandError.sMetsSearchCode) > 0 THEN
	sRejectReasonFSS := stCaseRejectReasons.stOuterBrandError.sFssSendCode;

ELSIF FIND(sRejectReasonME, stCaseRejectReasons.stCaseLabelBrandCodeError.sMetsSearchCode) > 0 THEN
	sRejectReasonFSS := stCaseRejectReasons.stCaseLabelBrandCodeError.sFssSendCode;

ELSE
	sRejectReasonFSS := stCaseRejectReasons.stUnknownCaseReject.sFssSendCode;
END_IF

F_CASE_GetRejectReasonFSS := sRejectReasonFSS;

END_FUNCTION

// ---- POUs/METS/Common LIB/06_KPI LIB/ClearStatistic/FB_KPI_ClearCameraInspection.TcPOU
FUNCTION_BLOCK FB_KPI_ClearCameraInspection
VAR_INPUT
	bExecute				: BOOL;
	stCTDateTime			: ST_SYSTEM_DateTime;	(* CaseTrace date/time structure *)
	sProductionSite		: STRING(4);
	sPCM				: STRING(4);
END_VAR
VAR_IN_OUT

	stPCMStatus			: ST_PCM_Status;
	stMetsCameras			: ST_NOVRAM_METS_Cameras;

END_VAR
VAR_OUTPUT
	bDone				: BOOL;
END_VAR
VAR
	fbExecute 			: R_TRIG;
	bTimerFlag			: BOOL;
	tofDoneTimer			: TOF;

	nCounter				: INT;
END_VAR

(* rising edge of bExecute *)
fbExecute(CLK:= bExecute);

bTimerFlag:=FALSE;

IF fbExecute.Q THEN

	nCounter := nCounter +1;

	MEMSET(ADR(stMetsCameras), 16#00, SIZEOF(stMetsCameras));

	stMetsCameras.MachineID.ProductionSite 	:= sProductionSite;
	stMetsCameras.MachineID.ProductionLine	:= sPCM;
	stMetsCameras.StartDateTime 				:=  F_SYSTEM_SystemTimeAsISO8601(stCTDateTime.sSystemTime, stCTDateTime.sUTCTimeZoneOffset );
	stMetsCameras.CodingAndTrackingMode 	:= stPCMStatus.nOpMode;

	bTimerFlag:=TRUE;
END_IF

tofDoneTimer(IN:=bTimerFlag,PT:=t#5s, Q=>bDone);

END_FUNCTION_BLOCK

// ---- POUs/METS/Common LIB/06_KPI LIB/ClearStatistic/FB_KPI_ClearExtCSStatistic.TcPOU
FUNCTION_BLOCK FB_KPI_ClearExtCSStatistic
VAR_INPUT
	bExecute				: BOOL;
	stCTDateTime			: ST_SYSTEM_DateTime;	(* CaseTrace date/time structure *)
	sProductionSite		: STRING(4);
	sPCM					: STRING(4);
END_VAR
VAR_IN_OUT
	stPCMStatus						: ST_PCM_Status;
	(*stCaseContentValidEfficiency		: ST_KPI_InspectionEfficency;
	stCaseLableValidEfficiency		: ST_KPI_InspectionEfficency;*)
	stCasePackerSignals				: ST_NOVRAM_METS_DualInputs;
	stCaseInspactionLog				: ST_NOVRAM_METS_CaseInspactionLog;
END_VAR
VAR_OUTPUT
	bDone				: BOOL;
END_VAR
VAR
	fbExecute 			: R_TRIG;
	bTimerFlag			: BOOL;
	tofDoneTimer			: TOF;

	nCounter				: INT;
END_VAR

(* rising edge of bExecute *)
fbExecute(CLK:= bExecute);

bTimerFlag:=FALSE;

IF fbExecute.Q THEN

	nCounter := nCounter +1;

(*	MEMSET(ADR(stCaseContentValidEfficiency), 16#00, SIZEOF(stCaseContentValidEfficiency));
	MEMSET(ADR(stCaseLableValidEfficiency), 16#00, SIZEOF(stCaseLableValidEfficiency));*)

	MEMSET(ADR(stCasePackerSignals), 16#00, SIZEOF(stCasePackerSignals));
	MEMSET(ADR(stCaseInspactionLog), 16#00, SIZEOF(stCaseInspactionLog));


	stCasePackerSignals.MachineID.ProductionSite	 := sProductionSite;
	stCasePackerSignals.MachineID.ProductionLine	:= sPCM;
	stCasePackerSignals.StartDateTime 				:=  F_SYSTEM_SystemTimeAsISO8601(stCTDateTime.sSystemTime, stCTDateTime.sUTCTimeZoneOffset );
	stCasePackerSignals.CodingAndTrackingMode	 	:=stPCMStatus.nOpMode;

	stCaseInspactionLog.MachineID.ProductionSite 	:= sProductionSite;
	stCaseInspactionLog.MachineID.ProductionLine	:= sPCM;
	stCaseInspactionLog.StartDateTime 				:=  F_SYSTEM_SystemTimeAsISO8601(stCTDateTime.sSystemTime, stCTDateTime.sUTCTimeZoneOffset );
	stCaseInspactionLog.CodingAndTrackingMode		:= stPCMStatus.nOpMode;
	stCaseInspactionLog.nPacksPerCase  			:= stPCMStatus.nPacksPerCase;
	stCaseInspactionLog.nOutersPerCase			:= stPCMStatus.nOutersPerCase;

	bTimerFlag:=TRUE;
END_IF

tofDoneTimer(IN:=bTimerFlag,PT:=t#5s, Q=>bDone);

END_FUNCTION_BLOCK

// ---- POUs/METS/Common LIB/06_KPI LIB/ClearStatistic/FB_KPI_ClearExtOUTStatistic.TcPOU
FUNCTION_BLOCK FB_KPI_ClearExtOUTStatistic
VAR_INPUT
	bExecute				: BOOL;
END_VAR
VAR_IN_OUT
	stOutersProcessing				: ST_KPI_OutersProcessing;
	aConfirmCodeEfficiency			: ARRAY[1..2] OF ST_KPI_CodePos;
	stPackConfirmationEfficiency		: ST_KPI_InspectionEfficency;
	aValidCodeEfficiency			: ARRAY[1..2] OF ST_KPI_CodePos;
	stOuterValidationEfficiency		: ST_KPI_InspectionEfficency;
END_VAR
VAR_OUTPUT
	bDone				: BOOL;
END_VAR
VAR
	fbExecute 			: R_TRIG;
	bTimerFlag			: BOOL;
	tofDoneTimer			: TOF;

	nCounter				: INT;
END_VAR

(* rising edge of bExecute *)
fbExecute(CLK:= bExecute);

bTimerFlag:=FALSE;

IF fbExecute.Q THEN

	nCounter := nCounter +1;

	stOutersProcessing.AtValidationCamera		:= 0;
	stOutersProcessing.AtConfimrationCamera	:= 0;
	MEMSET(ADR(aConfirmCodeEfficiency), 16#00, SIZEOF(aConfirmCodeEfficiency));
	MEMSET(ADR(stPackConfirmationEfficiency), 16#00, SIZEOF(stPackConfirmationEfficiency));
	MEMSET(ADR(aValidCodeEfficiency), 16#00, SIZEOF(aValidCodeEfficiency));
	MEMSET(ADR(stOuterValidationEfficiency), 16#00, SIZEOF(stOuterValidationEfficiency));

	bTimerFlag:=TRUE;
END_IF

tofDoneTimer(IN:=bTimerFlag,PT:=t#5s, Q=>bDone);

END_FUNCTION_BLOCK

// ---- POUs/METS/Common LIB/06_KPI LIB/ClearStatistic/FB_KPI_ClearExtPKStatistic.TcPOU
FUNCTION_BLOCK FB_KPI_ClearExtPKStatistic
VAR_INPUT
	bExecute				: BOOL;

END_VAR
VAR_IN_OUT
	stOutersProcessing				: ST_KPI_OutersProcessing;
	aPacksRead					: ARRAY[0..cMAX_PACKS_PER_OUTER] OF UDINT;
	aPackPosEfficiency				: ARRAY[1..cMAX_PACKS_PER_OUTER] OF ST_KPI_CodePos;
END_VAR
VAR_OUTPUT
	bDone				: BOOL;
END_VAR
VAR
	fbExecute 			: R_TRIG;
	bTimerFlag			: BOOL;
	tofDoneTimer			: TOF;

	nCounter				: INT;
END_VAR

(* rising edge of bExecute *)
fbExecute(CLK:= bExecute);

bTimerFlag:=FALSE;

IF fbExecute.Q THEN

	nCounter := nCounter +1;

	stOutersProcessing.AtPackAggregCameras	:= 0;
	MEMSET(ADR(aPacksRead), 16#00, SIZEOF(aPacksRead));
	MEMSET(ADR(aPackPosEfficiency), 16#00, SIZEOF(aPackPosEfficiency));

	bTimerFlag:=TRUE;
END_IF

tofDoneTimer(IN:=bTimerFlag,PT:=t#5s, Q=>bDone);

END_FUNCTION_BLOCK

// ---- POUs/METS/Common LIB/06_KPI LIB/ClearStatistic/FB_KPI_ClearFrontScreenStatistic.TcPOU
FUNCTION_BLOCK FB_KPI_ClearFrontScreenStatistic
VAR_INPUT
	bExecute				: BOOL;
	stCTDateTime			: ST_SYSTEM_DateTime;	(* CaseTrace date/time structure *)
	sProductionSite		: STRING(4);
	sPCM				: STRING(4);
END_VAR
VAR_IN_OUT

	stPCMStatus			: ST_PCM_Status;
	stMetsEfficiency		: ST_NOVRAM_METS_Inspection;
	stBarGraph			: ST_HMI_BarGraph;

END_VAR
VAR_OUTPUT
	bDone				: BOOL;
END_VAR
VAR
	fbExecute 			: R_TRIG;
	bTimerFlag			: BOOL;
	tofDoneTimer			: TOF;

	nCounter				: INT;
END_VAR

(* rising edge of bExecute *)
fbExecute(CLK:= bExecute);

bTimerFlag:=FALSE;

IF fbExecute.Q THEN

	nCounter := nCounter +1;


